// get unit number ----------------------------------------------------------
      L     DB1120.DBW    0;
      T     #UnitNo;

// communication ------------------------------------------------------------
      UC    FB  1125; // WT12Com

NETWORK
TITLE =Sequence organisation

      CLR   ;
      =     M    122.2;

// CIP Counter
      CALL FC    29 (
           UnitNo                   := #UnitNo,
           Value                    := DB1125.DBD   54,
           Enable                   := TRUE,
           Down                     := FALSE,
           OriginDetect             := 0.000000e+000,
           MaxDiffPS                := 1.000000e+000,
           SFMRec                   := DB1121.Seq.SFM[15],
           ValueOld                 := DB1121.DBD 1418);

// sequencer ----------------------------------------------------------------
      A     DB1123.DBX   43.1;
      S     DB1123.DBX   97.3;

      CALL FC    40 (
           UnitNo                   := #UnitNo);

END_FUNCTION_BLOCK

FUNCTION_BLOCK FB 1130
TITLE =U013: Wassertank 13
FAMILY : BOTEC_F1
NAME : U013A
VERSION : 2.1


VAR_TEMP
  EStopOK : BOOL ;	//auxiliary flag
  CIP : BOOL ;	//CIP Program Selected
  xTmp : BOOL ;	//Temporary Bool(free for general use)
  DummyBool : BOOL ;	//Temporary Bool(free for general use)
  UnitNo : INT ;	//unit number
  UnitFB : INT ;	//unit expansion FB number
  rTmp : REAL ;	//Temporary REAL (free for general use)
  iTmp : INT ;	//Temporary INT (free for general use)
  DummyInt : INT ;	//Temporary INT (free for general use)
  dTmp : DINT ;	//Temporary DINT (free for general use)
END_VAR
BEGIN
NETWORK
TITLE =general

      CLR   ;
      =     #xTmp;
      =     #EStopOK;

      L     DB1130.DBW    0;
      T     #UnitNo;
      L     DB1130.DBW    2;
      T     #UnitFB;

NETWORK
TITLE =analog inputs

      NOP   0;
// LI_T13 AnI 001 Niveau Tank 13
      CALL FC    24 (
           UnitNo                   := #UnitNo,
           AnIRec                   := DB2133.LI_T13,
           ValPer                   := DB302.DBW   88);

NETWORK
TITLE =Universal value

      NOP   0;
// unv001 UnV 001 Process Status
      CALL FC    27 (
           UnitNo                   := #UnitNo,
           UnVRec                   := DB2135.unv001,
           ValExt                   := DB2135.DBD  234);

// unv002 UnV 002 Universal Value 02
      CALL FC    27 (
           UnitNo                   := #UnitNo,
           UnVRec                   := DB2135.unv002,
           ValExt                   := DB2135.DBD  362);

// unv003 UnV 003 Universal Value 03
      CALL FC    27 (
           UnitNo                   := #UnitNo,
           UnVRec                   := DB2135.unv003,
           ValExt                   := DB2135.DBD  490);

NETWORK
TITLE =special inputs

      NOP   0;
// LS_LLL_T13 SpI 001 LS- Tank 13
      CALL FC    14 (
           UnitNo                   := #UnitNo,
           SpIRec                   := DB2131.LS_LLL_T13,
           SpIBit                   := I     50.0);

// LS_HL_T13 SpI 002 LS+ Tank 13
      CALL FC    14 (
           UnitNo                   := #UnitNo,
           SpIRec                   := DB2131.LS_HL_T13,
           SpIBit                   := I     49.6);

// GOA_T13_ML SpI 003 Mannloch Tank 13
      CALL FC    14 (
           UnitNo                   := #UnitNo,
           SpIRec                   := DB2131.GOA_T13_ML,
           SpIBit                   := I     49.5);

// GOA_T13_VV SpI 004 Vacuumventil Tank 13
      CALL FC    14 (
           UnitNo                   := #UnitNo,
           SpIRec                   := DB2131.GOA_T13_VV,
           SpIBit                   := I     49.4);

// LS_LL_T13 SpI 005 LS/ Tank 13
      CALL FC    14 (
           UnitNo                   := #UnitNo,
           SpIRec                   := DB2131.LS_LL_T13,
           SpIBit                   := I     49.7);

// RM_NI_T13_K4_AUF SpI 006
      CALL FC    14 (
           UnitNo                   := #UnitNo,
           SpIRec                   := DB2131.RM_NI_T13_K4_AUF,
           SpIBit                   := I     49.2);

// RM_NI_T13_K4_ZU SpI 007
      CALL FC    14 (
           UnitNo                   := #UnitNo,
           SpIRec                   := DB2131.RM_NI_T13_K4_ZU,
           SpIBit                   := I     49.3);

// RM_NI_T13_K2 SpI 008
      CALL FC    14 (
           UnitNo                   := #UnitNo,
           SpIRec                   := DB2131.RM_NI_T13_K2,
           SpIBit                   := I     49.0);

// RM_NI_T13_K3 SpI 010
      CALL FC    14 (
           UnitNo                   := #UnitNo,
           SpIRec                   := DB2131.RM_NI_T13_K3,
           SpIBit                   := I     49.1);

// LABOR_FREIG_T13 SpI 011 SCHLUESSELSCHALTER LABOR
      CALL FC    14 (
           UnitNo                   := #UnitNo,
           SpIRec                   := DB2131.LABOR_FREIG_T13,
           SpIBit                   := I    259.5);

NETWORK
TITLE =messages

      NOP   0;
// msg001 Msg 001 Message 01
      CALL FC    16 (
           UnitNo                   := #UnitNo,
           MsgRec                   := DB2137.msg001,
           MsgBit                   := DB2137.DBX   82.7);

// msg002 Msg 002 Message 02
      CALL FC    16 (
           UnitNo                   := #UnitNo,
           MsgRec                   := DB2137.msg002,
           MsgBit                   := DB2137.DBX  142.7);

NETWORK
TITLE =unit supply

      UC    FB [#UnitFB];

NETWORK
TITLE =T13_A10
// Act 005
// Box           : Ventilinsel 2
// Input address : I317.4
// Output address: Q317.4
      CALL FC    70 (
           UnitNo                   := #UnitNo,
           ActRec                   := DB2130.T13_A10,
           Typ                      := 1,
           FBa                      := #xTmp,
           FBa2                     := I    317.4,
           Out                      := Q    317.4);

NETWORK
TITLE =T13_A9
// Act 006
// Box           : Ventilinsel 2
// Input address : I319.4
// Output address: Q319.4
      CALL FC    70 (
           UnitNo                   := #UnitNo,
           ActRec                   := DB2130.T13_A9,
           Typ                      := 1,
           FBa                      := #xTmp,
           FBa2                     := I    319.4,
           Out                      := Q    319.4);

NETWORK
TITLE =T13_A12
// Act 007
// Box           : Ventilinsel 2
// Input address : I321.4
// Output address: Q321.4
      CALL FC    70 (
           UnitNo                   := #UnitNo,
           ActRec                   := DB2130.T13_A12,
           Typ                      := 1,
           FBa                      := #xTmp,
           FBa2                     := I    321.4,
           Out                      := Q    321.4);

NETWORK
TITLE =T13_A7
// Act 008
// Box           : Ventilinsel 2
// Input address : I323.4
// Output address: Q323.4
      CALL FC    70 (
           UnitNo                   := #UnitNo,
           ActRec                   := DB2130.T13_A7,
           Typ                      := 1,
           FBa                      := #xTmp,
           FBa2                     := I    323.4,
           Out                      := Q    323.4);

NETWORK
TITLE =T13_A8
// Act 009
// Box           : Ventilinsel 3
// Input address : I325.4
// Output address: Q325.4
      CALL FC    70 (
           UnitNo                   := #UnitNo,
           ActRec                   := DB2130.T13_A8,
           Typ                      := 1,
           FBa                      := #xTmp,
           FBa2                     := I    325.4,
           Out                      := Q    325.4);

NETWORK
TITLE =T13_A5
// Act 010
// Box           : Ventilinsel 3
// Input address : I327.4
// Output address: Q327.4
      CALL FC    70 (
           UnitNo                   := #UnitNo,
           ActRec                   := DB2130.T13_A5,
           Typ                      := 1,
           FBa                      := #xTmp,
           FBa2                     := I    327.4,
           Out                      := Q    327.4);

NETWORK
TITLE =T13_A11
// Act 011
// Box           : Ventilinsel 3
// Input address : I329.4
// Output address: Q329.4
      CALL FC    70 (
           UnitNo                   := #UnitNo,
           ActRec                   := DB2130.T13_A11,
           Typ                      := 1,
           FBa                      := #xTmp,
           FBa2                     := I    329.4,
           Out                      := Q    329.4);

NETWORK
TITLE =T13_A14
// Act 012
// Box           : Ventilinsel 4
// Input address : I331.4
// Output address: Q331.4
      CALL FC    70 (
           UnitNo                   := #UnitNo,
           ActRec                   := DB2130.T13_A14,
           Typ                      := 1,
           FBa                      := #xTmp,
           FBa2                     := I    331.4,
           Out                      := Q    331.4);

NETWORK
TITLE =T13_A15
// Act 013
// Box           : Ventilinsel 4
// Input address : I333.4
// Output address: Q333.4
      CALL FC    70 (
           UnitNo                   := #UnitNo,
           ActRec                   := DB2130.T13_A15,
           Typ                      := 0,
           FBa                      := #xTmp,
           FBa2                     := I    333.4,
           Out                      := Q    333.4);

NETWORK
TITLE =T13_RR1
// Act 014
// Box           : Ventilinsel 4
// Input address : I335.4
// Output address: Q335.4
      CALL FC    70 (
           UnitNo                   := #UnitNo,
           ActRec                   := DB2130.T13_RR1,
           Typ                      := 1,
           FBa                      := #xTmp,
           FBa2                     := I    335.4,
           Out                      := Q    335.4);

NETWORK
TITLE =RV1_T13
// Act 015
// Box           : Ventilinsel 1
// Input address : I10.4
// Output address: Q10.4
      CALL FC    70 (
           UnitNo                   := #UnitNo,
           ActRec                   := DB2130.RV1_T13,
           Typ                      := 1,
           FBa                      := #xTmp,
           FBa2                     := I     10.4,
           Out                      := Q     10.4);

NETWORK
TITLE =B6F_T13
// Act 016
// Box           : Ventilinsel 1
// Input address : I10.5
// Output address: Q10.5
      CALL FC    70 (
           UnitNo                   := #UnitNo,
           ActRec                   := DB2130.B6F_T13,
           Typ                      := 1,
           FBa                      := #xTmp,
           FBa2                     := I     10.5,
           Out                      := Q     10.5);

NETWORK
TITLE =H6F_T13
// Act 017
// Box           : Ventilinsel 1
// Input address : I10.6
// Output address: Q10.6
      CALL FC    70 (
           UnitNo                   := #UnitNo,
           ActRec                   := DB2130.H6F_T13,
           Typ                      := 1,
           FBa                      := #xTmp,
           FBa2                     := I     10.6,
           Out                      := Q     10.6);

NETWORK
TITLE =J6F_T13
// Act 018
// Box           : Ventilinsel 1
// Input address : I10.7
// Output address: Q10.7
      CALL FC    70 (
           UnitNo                   := #UnitNo,
           ActRec                   := DB2130.J6F_T13,
           Typ                      := 1,
           FBa                      := #xTmp,
           FBa2                     := I     10.7,
           Out                      := Q     10.7);

NETWORK
TITLE =L6F_T13
// Act 019
// Box           : Ventilinsel 1
// Input address : I11.0
// Output address: Q11.0
      CALL FC    70 (
           UnitNo                   := #UnitNo,
           ActRec                   := DB2130.L6F_T13,
           Typ                      := 1,
           FBa                      := #xTmp,
           FBa2                     := I     11.0,
           Out                      := Q     11.0);

NETWORK
TITLE =A_T13
// Act 022
// Box           : Ventilinsel 1
// Input address : I11.3
// Output address: Q11.3
      CALL FC    70 (
           UnitNo                   := #UnitNo,
           ActRec                   := DB2130.A_T13,
           Typ                      := 1,
           FBa                      := #xTmp,
           FBa2                     := I     11.3,
           Out                      := Q     11.3);

NETWORK
TITLE =B_T13
// Act 023
// Box           : Ventilinsel 1
// Input address : I11.4
// Output address: Q11.4
      CALL FC    70 (
           UnitNo                   := #UnitNo,
           ActRec                   := DB2130.B_T13,
           Typ                      := 1,
           FBa                      := #xTmp,
           FBa2                     := I     11.4,
           Out                      := Q     11.4);

NETWORK
TITLE =RW5_T13
// Act 026
// Box           : Ventilinsel 1
// Input address : I11.6
// Output address: Q11.6
      CALL FC    70 (
           UnitNo                   := #UnitNo,
           ActRec                   := DB2130.RW5_T13,
           Typ                      := 1,
           FBa                      := #xTmp,
           FBa2                     := I     11.6,
           Out                      := Q     11.6);

NETWORK
TITLE =RW6_T13
// Act 027
// Box           : Ventilinsel 1
// Input address : I11.7
// Output address: Q11.7
      CALL FC    70 (
           UnitNo                   := #UnitNo,
           ActRec                   := DB2130.RW6_T13,
           Typ                      := 1,
           FBa                      := #xTmp,
           FBa2                     := I     11.7,
           Out                      := Q     11.7);

NETWORK
TITLE =VVT13  Vacuumventil Tank 13
// Act 028
// Box           : VST1-9
// Output address: Q160.2
      CALL FC    70 (
           UnitNo                   := #UnitNo,
           ActRec                   := DB2130.VVT13,
           Typ                      := 0,
           FBa                      := #xTmp,
           FBa2                     := #xTmp,
           Out                      := Q    160.2);

NETWORK
TITLE =VR_T13
// Act 029
// Box           : Ventilinsel 1
// Output address: Q11.5
      CALL FC    70 (
           UnitNo                   := #UnitNo,
           ActRec                   := DB2130.VR_T13,
           Typ                      := 0,
           FBa                      := #xTmp,
           FBa2                     := #xTmp,
           Out                      := Q     11.5);

NETWORK
TITLE =ML_LABORFREIGABE_T13
// Act 031
// Box           : LT-CIP
// Output address: Q259.5
      CALL FC    70 (
           UnitNo                   := #UnitNo,
           ActRec                   := DB2130.ML_LABORFREIGABE_T13,
           Typ                      := 0,
           FBa                      := #xTmp,
           FBa2                     := #xTmp,
           Out                      := Q    259.5);

END_FUNCTION_BLOCK

FUNCTION_BLOCK FB 1131
TITLE =U013: Water Tank 13
FAMILY : BOTEC_F1
NAME : UniE
VERSION : 1.2


VAR_TEMP
  CIP : BOOL ;	//CIP active
  UNIM : BOOL ;	//Unit Not In Maintenance
  GenRel : BOOL ;	//general OK (emergency and maintenance OK)
  EStopOK : BOOL ;	//emergency OK
  UnitNo : INT ;	//unit number
  xTmp : BOOL ;	//Temporary Bool
  iTmp : INT ;	//Temporary INT
  rTmp : REAL ;	//Temporary REAL
  dTmp : DINT ;	//Temporary DINT (free for general use)
  RetValInt : INT ;	//return value
END_VAR
BEGIN
NETWORK
TITLE =General

      SET   ;
// Simulation ---------------------------------------------------------------
      A     DB1131.DBX 1357.7;
      CC    FB  1139; // "WT13Sim"
      A     DB1131.DBX   17.3;
      =     DB1131.DBX 1357.7; //Help bit for simulation

// get unit number ----------------------------------------------------------
      L     DB1130.DBW    0;
      T     #UnitNo;

// communication ------------------------------------------------------------
      UC    FB  1135; // WT13Com

NETWORK
TITLE =Sequence organisation

      CLR   ;
      =     M    122.2;

// CIP Counter
      CALL FC    29 (
           UnitNo                   := #UnitNo,
           Value                    := DB1135.DBD   54,
           Enable                   := TRUE,
           Down                     := FALSE,
           OriginDetect             := 0.000000e+000,
           MaxDiffPS                := 1.000000e+000,
           SFMRec                   := DB1131.Seq.SFM[15],
           ValueOld                 := DB1131.DBD 1418);

// sequencer ----------------------------------------------------------------
      A     DB1133.DBX   43.1;
      S     DB1133.DBX   97.3;

      CALL FC    40 (
           UnitNo                   := #UnitNo);

END_FUNCTION_BLOCK

FUNCTION_BLOCK FB 1210
TITLE =U021: Brunnen Transfer VE1
FAMILY : BOTEC_F1
NAME : U021A
VERSION : 2.1


VAR_TEMP
  EStopOK : BOOL ;	//auxiliary flag
  CIP : BOOL ;	//CIP Program Selected
  xTmp : BOOL ;	//Temporary Bool(free for general use)
  DummyBool : BOOL ;	//Temporary Bool(free for general use)
  UnitNo : INT ;	//unit number
  UnitFB : INT ;	//unit expansion FB number
  rTmp : REAL ;	//Temporary REAL (free for general use)
  iTmp : INT ;	//Temporary INT (free for general use)
  DummyInt : INT ;	//Temporary INT (free for general use)
  dTmp : DINT ;	//Temporary DINT (free for general use)
END_VAR
BEGIN
NETWORK
TITLE =general

      CLR   ;
      =     #xTmp;
      =     #EStopOK;

      L     DB1210.DBW    0;
      T     #UnitNo;
      L     DB1210.DBW    2;
      T     #UnitFB;

NETWORK
TITLE =analog inputs

      NOP   0;
// C_AnI01 AnI 001 spare
      CALL FC    24 (
           UnitNo                   := #UnitNo,
           AnIRec                   := DB2213.C_AnI01,
           ValPer                   := #DummyInt);

// C_AnI002 AnI 002 spare
      CALL FC    24 (
           UnitNo                   := #UnitNo,
           AnIRec                   := DB2213.C_AnI002,
           ValPer                   := #DummyInt);

// AnI03 AnI 003 spare
      CALL FC    24 (
           UnitNo                   := #UnitNo,
           AnIRec                   := DB2213.AnI03,
           ValPer                   := #DummyInt);

NETWORK
TITLE =Universal value

      NOP   0;
// unv001 UnV 001 Process Status
      CALL FC    27 (
           UnitNo                   := #UnitNo,
           UnVRec                   := DB2215.unv001,
           ValExt                   := DB2215.DBD  234);

// unv002 UnV 002 Universal Value 02
      CALL FC    27 (
           UnitNo                   := #UnitNo,
           UnVRec                   := DB2215.unv002,
           ValExt                   := DB2215.DBD  362);

// unv003 UnV 003 Universal Value 03
      CALL FC    27 (
           UnitNo                   := #UnitNo,
           UnVRec                   := DB2215.unv003,
           ValExt                   := DB2215.DBD  490);

// unv004 UnV 004 Universal Value 04
      CALL FC    27 (
           UnitNo                   := #UnitNo,
           UnVRec                   := DB2215.unv004,
           ValExt                   := DB2215.DBD  618);

NETWORK
TITLE =special inputs

      NOP   0;
// NI_VP1_Br2a_VE1 SpI 001 Paneel VP1 Brunnen 2a -> VE1
      CALL FC    14 (
           UnitNo                   := #UnitNo,
           SpIRec                   := DB2211.NI_VP1_Br2a_VE1,
           SpIBit                   := I     80.1);

// NI_VP1_Br2b_VE1 SpI 002 Paneel VP1 Brunnen 2b -> VE1
      CALL FC    14 (
           UnitNo                   := #UnitNo,
           SpIRec                   := DB2211.NI_VP1_Br2b_VE1,
           SpIBit                   := I     80.2);

// NI_VP1_Br3_VE1 SpI 003 Paneel VP1 Brunnen 3 -> VE1
      CALL FC    14 (
           UnitNo                   := #UnitNo,
           SpIRec                   := DB2211.NI_VP1_Br3_VE1,
           SpIBit                   := I     80.4);

// NI_VP1_Br7_VE1 SpI 004 Paneel VP1 Brunnen 7 -> VE1
      CALL FC    14 (
           UnitNo                   := #UnitNo,
           SpIRec                   := DB2211.NI_VP1_Br7_VE1,
           SpIBit                   := I     80.3);

NETWORK
TITLE =messages

      NOP   0;
// msg001 Msg 001 Message 01
      CALL FC    16 (
           UnitNo                   := #UnitNo,
           MsgRec                   := DB2217.msg001,
           MsgBit                   := DB2217.DBX   82.7);

// msg002 Msg 002 Message 02
      CALL FC    16 (
           UnitNo                   := #UnitNo,
           MsgRec                   := DB2217.msg002,
           MsgBit                   := DB2217.DBX  142.7);

// msg003 Msg 003 Message 03
      CALL FC    16 (
           UnitNo                   := #UnitNo,
           MsgRec                   := DB2217.msg003,
           MsgBit                   := DB2217.DBX  202.7);

NETWORK
TITLE =controllers

      NOP   0;
// PID01 PID 001 spare
      CALL FC    55 (
           UnitNo                   := #UnitNo,
           PIDRec                   := DB2216.PID01,
           SpExt                    := DB2216.DBD  234,
           PVal                     := DB2216.DBD  254,
           OPer                     := #DummyInt);

NETWORK
TITLE =unit supply

      UC    FB [#UnitFB];

NETWORK
TITLE =RW6_G1  Gullyventil RW6
// Act 001
// Box           : VS2-BB
// Input address : I310.4
// Output address: Q310.4
      CALL FC    70 (
           UnitNo                   := #UnitNo,
           ActRec                   := DB2210.RW6_G1,
           Typ                      := 1,
           FBa                      := #xTmp,
           FBa2                     := I    310.4,
           Out                      := Q    310.4);

NETWORK
TITLE =VE1V1  VE1V1 --> Chriwa
// Act 002
// Box           : VS2-BB
// Input address : I310.5
// Output address: Q310.5
      CALL FC    70 (
           UnitNo                   := #UnitNo,
           ActRec                   := DB2210.VE1V1,
           Typ                      := 23,
           FBa                      := I    310.5,
           FBa2                     := #xTmp,
           Out                      := Q    310.5);

NETWORK
TITLE =VE1V2  VE1V2 Gully
// Act 003
// Box           : VS2-BB
// Input address : I310.6
// Output address: Q310.6
      CALL FC    70 (
           UnitNo                   := #UnitNo,
           ActRec                   := DB2210.VE1V2,
           Typ                      := 1,
           FBa                      := #xTmp,
           FBa2                     := I    310.6,
           Out                      := Q    310.6);

END_FUNCTION_BLOCK

FUNCTION_BLOCK FB 1211
TITLE =U021: Well Transfer VE1
FAMILY : BOTEC_F1
NAME : UniE
VERSION : 1.2


VAR_TEMP
  CIP : BOOL ;	//CIP active
  UNIM : BOOL ;	//Unit Not In Maintenance
  GenRel : BOOL ;	//general OK (emergency and maintenance OK)
  EStopOK : BOOL ;	//emergency OK
  UnitNo : INT ;	//unit number
  xTmp : BOOL ;	//Temporary Bool
  iTmp : INT ;	//Temporary INT
  rTmp : REAL ;	//Temporary REAL
  dTmp : DINT ;	//Temporary DINT (free for general use)
  RetValInt : INT ;	//return value
END_VAR
BEGIN
NETWORK
TITLE =General

      SET   ;
// Simulation ---------------------------------------------------------------
      A     DB1211.DBX 1357.7;
      CC    FB  1219; // "U021Sim"
      A     DB1211.DBX   17.3;
      =     DB1211.DBX 1357.7; //Help bit for simulation

// get unit number ----------------------------------------------------------
      L     DB1210.DBW    0;
      T     #UnitNo;

// communication ------------------------------------------------------------
      UC    FB  1215; // U021Com

NETWORK
TITLE =Sequence organisation

      CLR   ;
      =     M    122.2;


// Chriwa Status 1
      L     DB1381.DBD  482;
      T     DB1211.DBD  482;

// Chriwa Status 2
      L     DB1381.DBD  498;
      T     DB1211.DBD  498;

// sequencer ----------------------------------------------------------------
      A     DB1213.DBX   43.1;
      S     DB1213.DBX   97.3;

      CALL FC    40 (
           UnitNo                   := #UnitNo);

END_FUNCTION_BLOCK

FUNCTION_BLOCK FB 1220
TITLE =U022: Brunnen Transfer VE2
FAMILY : BOTEC_F1
NAME : U022A
VERSION : 2.1


VAR_TEMP
  EStopOK : BOOL ;	//auxiliary flag
  CIP : BOOL ;	//CIP Program Selected
  xTmp : BOOL ;	//Temporary Bool(free for general use)
  DummyBool : BOOL ;	//Temporary Bool(free for general use)
  UnitNo : INT ;	//unit number
  UnitFB : INT ;	//unit expansion FB number
  rTmp : REAL ;	//Temporary REAL (free for general use)
  iTmp : INT ;	//Temporary INT (free for general use)
  DummyInt : INT ;	//Temporary INT (free for general use)
  dTmp : DINT ;	//Temporary DINT (free for general use)
END_VAR
BEGIN
NETWORK
TITLE =general

      CLR   ;
      =     #xTmp;
      =     #EStopOK;

      L     DB1220.DBW    0;
      T     #UnitNo;
      L     DB1220.DBW    2;
      T     #UnitFB;

NETWORK
TITLE =analog inputs

      NOP   0;
// C_AnI01 AnI 001 spare
      CALL FC    24 (
           UnitNo                   := #UnitNo,
           AnIRec                   := DB2223.C_AnI01,
           ValPer                   := #DummyInt);

// C_AnI002 AnI 002 spare
      CALL FC    24 (
           UnitNo                   := #UnitNo,
           AnIRec                   := DB2223.C_AnI002,
           ValPer                   := #DummyInt);

// AnI03 AnI 003 spare
      CALL FC    24 (
           UnitNo                   := #UnitNo,
           AnIRec                   := DB2223.AnI03,
           ValPer                   := #DummyInt);

NETWORK
TITLE =Universal value

      NOP   0;
// unv001 UnV 001 Process Status
      CALL FC    27 (
           UnitNo                   := #UnitNo,
           UnVRec                   := DB2225.unv001,
           ValExt                   := DB2225.DBD  234);

// unv002 UnV 002 Universal Value 02
      CALL FC    27 (
           UnitNo                   := #UnitNo,
           UnVRec                   := DB2225.unv002,
           ValExt                   := DB2225.DBD  362);

// unv003 UnV 003 Universal Value 03
      CALL FC    27 (
           UnitNo                   := #UnitNo,
           UnVRec                   := DB2225.unv003,
           ValExt                   := DB2225.DBD  490);

// unv004 UnV 004 Universal Value 04
      CALL FC    27 (
           UnitNo                   := #UnitNo,
           UnVRec                   := DB2225.unv004,
           ValExt                   := DB2225.DBD  618);

NETWORK
TITLE =special inputs

      NOP   0;
// NI_VP1_Br2a_VE2 SpI 001 Paneel VP1 Brunnen 2a -> VE2
      CALL FC    14 (
           UnitNo                   := #UnitNo,
           SpIRec                   := DB2221.NI_VP1_Br2a_VE2,
           SpIBit                   := I     80.6);

// NI_VP1_Br2b_VE2 SpI 002 Paneel VP1 Brunnen 2b -> VE2
      CALL FC    14 (
           UnitNo                   := #UnitNo,
           SpIRec                   := DB2221.NI_VP1_Br2b_VE2,
           SpIBit                   := I     80.7);

// NI_VP1_Br3_VE2 SpI 003 Paneel VP1 Brunnen 3 -> VE2
      CALL FC    14 (
           UnitNo                   := #UnitNo,
           SpIRec                   := DB2221.NI_VP1_Br3_VE2,
           SpIBit                   := I     81.1);

// NI_VP1_Br7_VE2 SpI 004 Paneel VP1 Brunnen 7 -> VE2
      CALL FC    14 (
           UnitNo                   := #UnitNo,
           SpIRec                   := DB2221.NI_VP1_Br7_VE2,
           SpIBit                   := I     81.0);

NETWORK
TITLE =messages

      NOP   0;
// msg001 Msg 001 Message 01
      CALL FC    16 (
           UnitNo                   := #UnitNo,
           MsgRec                   := DB2227.msg001,
           MsgBit                   := DB2227.DBX   82.7);

// msg002 Msg 002 Message 02
      CALL FC    16 (
           UnitNo                   := #UnitNo,
           MsgRec                   := DB2227.msg002,
           MsgBit                   := DB2227.DBX  142.7);

// msg003 Msg 003 Message 03
      CALL FC    16 (
           UnitNo                   := #UnitNo,
           MsgRec                   := DB2227.msg003,
           MsgBit                   := DB2227.DBX  202.7);

NETWORK
TITLE =controllers

      NOP   0;
// PID01 PID 001 spare
      CALL FC    55 (
           UnitNo                   := #UnitNo,
           PIDRec                   := DB2226.PID01,
           SpExt                    := DB2226.DBD  234,
           PVal                     := DB2226.DBD  254,
           OPer                     := #DummyInt);

NETWORK
TITLE =unit supply

      UC    FB [#UnitFB];

NETWORK
TITLE =RW5_G1  Gullyventil RW5
// Act 001
// Box           : VS2-BB
// Input address : I310.3
// Output address: Q310.3
      CALL FC    70 (
           UnitNo                   := #UnitNo,
           ActRec                   := DB2220.RW5_G1,
           Typ                      := 1,
           FBa                      := #xTmp,
           FBa2                     := I    310.3,
           Out                      := Q    310.3);

NETWORK
TITLE =VE2V1  VE2V1 --> Chriwa
// Act 002
// Box           : VS2-BB
// Input address : I310.7
// Output address: Q310.7
      CALL FC    70 (
           UnitNo                   := #UnitNo,
           ActRec                   := DB2220.VE2V1,
           Typ                      := 23,
           FBa                      := I    310.7,
           FBa2                     := #xTmp,
           Out                      := Q    310.7);

NETWORK
TITLE =VE2V2  VE2V2 Gully
// Act 003
// Box           : VS2-BB
// Input address : I311.0
// Output address: Q311.0
      CALL FC    70 (
           UnitNo                   := #UnitNo,
           ActRec                   := DB2220.VE2V2,
           Typ                      := 1,
           FBa                      := #xTmp,
           FBa2                     := I    311.0,
           Out                      := Q    311.0);

END_FUNCTION_BLOCK

FUNCTION_BLOCK FB 1221
TITLE =U022: Well Transfer VE2
FAMILY : BOTEC_F1
NAME : UniE
VERSION : 1.2


VAR_TEMP
  CIP : BOOL ;	//CIP active
  UNIM : BOOL ;	//Unit Not In Maintenance
  GenRel : BOOL ;	//general OK (emergency and maintenance OK)
  EStopOK : BOOL ;	//emergency OK
  UnitNo : INT ;	//unit number
  xTmp : BOOL ;	//Temporary Bool
  iTmp : INT ;	//Temporary INT
  rTmp : REAL ;	//Temporary REAL
  dTmp : DINT ;	//Temporary DINT (free for general use)
  RetValInt : INT ;	//return value
END_VAR
BEGIN
NETWORK
TITLE =General

      SET   ;
// Simulation ---------------------------------------------------------------
      A     DB1221.DBX 1357.7;
      CC    FB  1229; // "U022Sim"
      A     DB1221.DBX   17.3;
      =     DB1221.DBX 1357.7; //Help bit for simulation

// get unit number ----------------------------------------------------------
      L     DB1220.DBW    0;
      T     #UnitNo;

// communication ------------------------------------------------------------
      UC    FB  1225; // U022Com

NETWORK
TITLE =Sequence organisation

      CLR   ;
      =     M    122.2;


// Chriwa Status 1
      L     DB1391.DBD  482;
      T     DB1221.DBD  482;

// Chriwa Status 2
      L     DB1391.DBD  498;
      T     DB1221.DBD  498;

// sequencer ----------------------------------------------------------------
      A     DB1223.DBX   43.1;
      S     DB1223.DBX   97.3;

      CALL FC    40 (
           UnitNo                   := #UnitNo);

END_FUNCTION_BLOCK

FUNCTION_BLOCK FB 1250
TITLE =U025: Well Transfer A
FAMILY : BOTEC_F1
NAME : UniA
VERSION : 2.1


VAR_TEMP
  EStopOK : BOOL ;	//auxiliary flag
  CIP : BOOL ;	//CIP Program Selected
  xTmp : BOOL ;	//Temporary Bool(free for general use)
  UnitNo : INT ;	//unit number
  UnitFB : INT ;	//unit expansion FB number
  rTmp : REAL ;	//Temporary REAL (free for general use)
  iTmp : INT ;	//Temporary INT (free for general use)
  dTmp : DINT ;	//Temporary DINT (free for general use)
END_VAR
BEGIN
NETWORK
TITLE =general

      CLR   ;
      =     #xTmp;
      =     #EStopOK;

      L     DB1250.DBW    0;
      T     #UnitNo;
      L     DB1250.DBW    2;
      T     #UnitFB;

NETWORK
TITLE =analog inputs

      NOP   0;
// C_AnI01 AnI 001 spare
      CALL FC    24 (
           UnitNo                   := #UnitNo,
           AnIRec                   := DB2253.C_AnI01,
           ValPer                   := #iTmp);

// QI_CO2_A_PH AnI 002
      CALL FC    24 (
           UnitNo                   := #UnitNo,
           AnIRec                   := DB2253.QI_CO2_A_PH,
           ValPer                   := IW   220);

// QI_CO2_A_pH_KOR AnI 003 pH Brunnen A mit Offset
      CALL FC    24 (
           UnitNo                   := #UnitNo,
           AnIRec                   := DB2253.QI_CO2_A_pH_KOR,
           ValPer                   := IW   552);

NETWORK
TITLE =Universal value

      NOP   0;
// unv001 UnV 001 Process Status
      CALL FC    27 (
           UnitNo                   := #UnitNo,
           UnVRec                   := DB2255.unv001,
           ValExt                   := DB2255.DBD  234);

// unv002 UnV 002 Universal Value 02
      CALL FC    27 (
           UnitNo                   := #UnitNo,
           UnVRec                   := DB2255.unv002,
           ValExt                   := DB2255.DBD  362);

// unv003 UnV 003 Universal Value 03
      CALL FC    27 (
           UnitNo                   := #UnitNo,
           UnVRec                   := DB2255.unv003,
           ValExt                   := DB2255.DBD  490);

// unv004 UnV 004 Universal Value 04
      CALL FC    27 (
           UnitNo                   := #UnitNo,
           UnVRec                   := DB2255.unv004,
           ValExt                   := DB2255.DBD  618);

NETWORK
TITLE =special inputs

      NOP   0;
// SpI01 SpI 001 spare
      CALL FC    14 (
           UnitNo                   := #UnitNo,
           SpIRec                   := DB2251.SpI01,
           SpIBit                   := #xTmp);

// SpI02 SpI 002 spare
      CALL FC    14 (
           UnitNo                   := #UnitNo,
           SpIRec                   := DB2251.SpI02,
           SpIBit                   := #xTmp);

// SpI03 SpI 003 spare
      CALL FC    14 (
           UnitNo                   := #UnitNo,
           SpIRec                   := DB2251.SpI03,
           SpIBit                   := #xTmp);

// SpI04 SpI 004 spare
      CALL FC    14 (
           UnitNo                   := #UnitNo,
           SpIRec                   := DB2251.SpI04,
           SpIBit                   := #xTmp);

NETWORK
TITLE =messages

      NOP   0;
// msg001 Msg 001 Message 01
      CALL FC    16 (
           UnitNo                   := #UnitNo,
           MsgRec                   := DB2257.msg001,
           MsgBit                   := DB2257.DBX   82.7);

// msg002 Msg 002 Message 02
      CALL FC    16 (
           UnitNo                   := #UnitNo,
           MsgRec                   := DB2257.msg002,
           MsgBit                   := DB2257.DBX  142.7);

// msg003 Msg 003 Message 03
      CALL FC    16 (
           UnitNo                   := #UnitNo,
           MsgRec                   := DB2257.msg003,
           MsgBit                   := DB2257.DBX  202.7);

NETWORK
TITLE =controllers

      NOP   0;
// CO2ARV1 PID 001 CO2 A RV1
      CALL FC    55 (
           UnitNo                   := #UnitNo,
           PIDRec                   := DB2256.CO2ARV1,
           SpExt                    := DB2256.DBD  234,
           PVal                     := DB2256.DBD  254,
           OPer                     := PQW  220);

NETWORK
TITLE =unit supply

      UC    FB [#UnitFB];

NETWORK
TITLE =A_G1  A_G1
// Act 001
// Box           : VS2-BB
// Output address: Q309.3
      CALL FC    70 (
           UnitNo                   := #UnitNo,
           ActRec                   := DB2250.A_G1,
           Typ                      := 1,
           FBa                      := #xTmp,
           FBa2                     := I    309.3,
           Out                      := Q    309.3);

NETWORK
TITLE =CO2_AV2  Ansteuerung AV2
// Act 002
// Box           : CO2 Dosierung
// Output address: Q61.7
      CALL FC    70 (
           UnitNo                   := #UnitNo,
           ActRec                   := DB2250.CO2_AV2,
           Typ                      := 0,
           FBa                      := #xTmp,
           FBa2                     := #xTmp,
           Out                      := Q     61.7);

NETWORK
TITLE =CO2_AV1  Ansteuerung AV1
// Act 003
// Box           : CO2 Dosierung
// Output address: Q60.7
      CALL FC    70 (
           UnitNo                   := #UnitNo,
           ActRec                   := DB2250.CO2_AV1,
           Typ                      := 0,
           FBa                      := #xTmp,
           FBa2                     := #xTmp,
           Out                      := Q     60.7);

NETWORK
TITLE =ARV1  CO2 A RV1
// Act 004
// Box           :
// Input address : #xtmp
// Output address: #xtmp
      CALL FC    70 (
           UnitNo                   := #UnitNo,
           ActRec                   := DB2250.ARV1,
           Typ                      := 4,
           FBa                      := #xTmp,
           FBa2                     := #xTmp,
           Out                      := #xTmp);

END_FUNCTION_BLOCK

FUNCTION_BLOCK FB 1251
TITLE =U025: Well Transfer A
FAMILY : BOTEC_F1
NAME : UniE
VERSION : 1.2


VAR_TEMP
  CIP : BOOL ;	//CIP active
  UNIM : BOOL ;	//Unit Not In Maintenance
  GenRel : BOOL ;	//general OK (emergency and maintenance OK)
  EStopOK : BOOL ;	//emergency OK
  UnitNo : INT ;	//unit number
  xTmp : BOOL ;	//Temporary Bool
  iTmp : INT ;	//Temporary INT
  rTmp : REAL ;	//Temporary REAL
  dTmp : DINT ;	//Temporary DINT (free for general use)
  RetValInt : INT ;	//return value
END_VAR
BEGIN
NETWORK
TITLE =General

      SET   ;
// Simulation ---------------------------------------------------------------
      A     DB1251.DBX 1357.7;
      CC    FB  1259; // "U025Sim"
      A     DB1251.DBX   17.3;
      =     DB1251.DBX 1357.7; //Help bit for simulation

// get unit number ----------------------------------------------------------
      L     DB1250.DBW    0;
      T     #UnitNo;

// communication ------------------------------------------------------------
      UC    FB  1255; // U025Com

NETWORK
TITLE =Sequence organisation

      CLR   ;
      =     M    122.2;

// sequencer ----------------------------------------------------------------
      A     DB1253.DBX   43.1;
      S     DB1253.DBX   97.3;

      CALL FC    40 (
           UnitNo                   := #UnitNo);

END_FUNCTION_BLOCK

FUNCTION_BLOCK FB 1260
TITLE =U026: Well Transfer B
FAMILY : BOTEC_F1
NAME : UniA
VERSION : 2.1


VAR_TEMP
  EStopOK : BOOL ;	//auxiliary flag
  CIP : BOOL ;	//CIP Program Selected
  xTmp : BOOL ;	//Temporary Bool(free for general use)
  UnitNo : INT ;	//unit number
  UnitFB : INT ;	//unit expansion FB number
  rTmp : REAL ;	//Temporary REAL (free for general use)
  iTmp : INT ;	//Temporary INT (free for general use)
  dTmp : DINT ;	//Temporary DINT (free for general use)
END_VAR
BEGIN
NETWORK
TITLE =general

      CLR   ;
      =     #xTmp;
      =     #EStopOK;

      L     DB1260.DBW    0;
      T     #UnitNo;
      L     DB1260.DBW    2;
      T     #UnitFB;

NETWORK
TITLE =analog inputs

      NOP   0;
// C_AnI01 AnI 001 spare
      CALL FC    24 (
           UnitNo                   := #UnitNo,
           AnIRec                   := DB2263.C_AnI01,
           ValPer                   := #iTmp);

// QI_CO2_B_PH AnI 002
      CALL FC    24 (
           UnitNo                   := #UnitNo,
           AnIRec                   := DB2263.QI_CO2_B_PH,
           ValPer                   := IW   222);

// AnI03 AnI 003 spare
      CALL FC    24 (
           UnitNo                   := #UnitNo,
           AnIRec                   := DB2263.AnI03,
           ValPer                   := #iTmp);

NETWORK
TITLE =Universal value

      NOP   0;
// unv001 UnV 001 Process Status
      CALL FC    27 (
           UnitNo                   := #UnitNo,
           UnVRec                   := DB2265.unv001,
           ValExt                   := DB2265.DBD  234);

// unv002 UnV 002 Universal Value 02
      CALL FC    27 (
           UnitNo                   := #UnitNo,
           UnVRec                   := DB2265.unv002,
           ValExt                   := DB2265.DBD  362);

// unv003 UnV 003 Universal Value 03
      CALL FC    27 (
           UnitNo                   := #UnitNo,
           UnVRec                   := DB2265.unv003,
           ValExt                   := DB2265.DBD  490);

// unv004 UnV 004 Universal Value 04
      CALL FC    27 (
           UnitNo                   := #UnitNo,
           UnVRec                   := DB2265.unv004,
           ValExt                   := DB2265.DBD  618);

NETWORK
TITLE =special inputs

      NOP   0;
// RM_NI_KF1_K1 SpI 001
      CALL FC    14 (
           UnitNo                   := #UnitNo,
           SpIRec                   := DB2261.RM_NI_KF1_K1,
           SpIBit                   := #xTmp);//"RM_NI_KF1_K1"

// RM_NI_KF1_K2 SpI 002
      CALL FC    14 (
           UnitNo                   := #UnitNo,
           SpIRec                   := DB2261.RM_NI_KF1_K2,
           SpIBit                   := #xTmp);//"RM_NI_KF1_K2"

// RM_NI_KF1_K3 SpI 003 PANEEL PTV1
      CALL FC    14 (
           UnitNo                   := #UnitNo,
           SpIRec                   := DB2261.RM_NI_KF1_K3,
           SpIBit                   := I     54.6);


// SpI04 SpI 004 spare
      CALL FC    14 (
           UnitNo                   := #UnitNo,
           SpIRec                   := DB2261.SpI04,
           SpIBit                   := #xTmp);

NETWORK
TITLE =messages

      NOP   0;
// msg001 Msg 001 Message 01
      CALL FC    16 (
           UnitNo                   := #UnitNo,
           MsgRec                   := DB2267.msg001,
           MsgBit                   := DB2267.DBX   82.7);

// msg002 Msg 002 Message 02
      CALL FC    16 (
           UnitNo                   := #UnitNo,
           MsgRec                   := DB2267.msg002,
           MsgBit                   := DB2267.DBX  142.7);

// msg003 Msg 003 Message 03
      CALL FC    16 (
           UnitNo                   := #UnitNo,
           MsgRec                   := DB2267.msg003,
           MsgBit                   := DB2267.DBX  202.7);

NETWORK
TITLE =controllers

      NOP   0;
// CO2BRV1 PID 001 CO2 B RV1
      CALL FC    55 (
           UnitNo                   := #UnitNo,
           PIDRec                   := DB2266.CO2BRV1,
           SpExt                    := DB2266.DBD  234,
           PVal                     := DB2266.DBD  254,
           OPer                     := PQW  222);

NETWORK
TITLE =unit supply

      UC    FB [#UnitFB];

NETWORK
TITLE =B_G1  B_G1
// Act 001
// Box           : VS2-BB
// Output address: Q309.4
      CALL FC    70 (
           UnitNo                   := #UnitNo,
           ActRec                   := DB2260.B_G1,
           Typ                      := 1,
           FBa                      := #xTmp,
           FBa2                     := I    309.4,
           Out                      := Q    309.4);

NETWORK
TITLE =CO2_BV2  Ansteuerung BV2
// Act 002
// Box           : CO2 Dosierung
// Output address: Q61.6
      CALL FC    70 (
           UnitNo                   := #UnitNo,
           ActRec                   := DB2260.CO2_BV2,
           Typ                      := 0,
           FBa                      := #xTmp,
           FBa2                     := #xTmp,
           Out                      := Q     61.6);

NETWORK
TITLE =CO2_BV1  Ansteuerung BV1
// Act 003
// Box           : CO2 Dosierung
// Output address: Q60.6
      CALL FC    70 (
           UnitNo                   := #UnitNo,
           ActRec                   := DB2260.CO2_BV1,
           Typ                      := 0,
           FBa                      := #xTmp,
           FBa2                     := #xTmp,
           Out                      := Q     60.6);

NETWORK
TITLE =BRV1  CO2 B RV1
// Act 004
// Box           :
// Input address : #xtmp
// Output address: #xtmp
      CALL FC    70 (
           UnitNo                   := #UnitNo,
           ActRec                   := DB2260.BRV1,
           Typ                      := 4,
           FBa                      := #xTmp,
           FBa2                     := #xTmp,
           Out                      := #xTmp);

END_FUNCTION_BLOCK

FUNCTION_BLOCK FB 1261
TITLE =U026: Well Transfer B
FAMILY : BOTEC_F1
NAME : UniE
VERSION : 1.2


VAR_TEMP
  CIP : BOOL ;	//CIP active
  UNIM : BOOL ;	//Unit Not In Maintenance
  GenRel : BOOL ;	//general OK (emergency and maintenance OK)
  EStopOK : BOOL ;	//emergency OK
  UnitNo : INT ;	//unit number
  xTmp : BOOL ;	//Temporary Bool
  iTmp : INT ;	//Temporary INT
  rTmp : REAL ;	//Temporary REAL
  dTmp : DINT ;	//Temporary DINT (free for general use)
  RetValInt : INT ;	//return value
END_VAR
BEGIN
NETWORK
TITLE =General

      SET   ;
// Simulation ---------------------------------------------------------------
      A     DB1261.DBX 1357.7;
      CC    FB  1269; // "U026Sim"
      A     DB1261.DBX   17.3;
      =     DB1261.DBX 1357.7; //Help bit for simulation

// get unit number ----------------------------------------------------------
      L     DB1260.DBW    0;
      T     #UnitNo;

// communication ------------------------------------------------------------
      UC    FB  1265; // U026Com

NETWORK
TITLE =Sequence organisation

      CLR   ;
      =     M    122.2;

// sequencer ----------------------------------------------------------------
      A     DB1263.DBX   43.1;
      S     DB1263.DBX   97.3;

      CALL FC    40 (
           UnitNo                   := #UnitNo);

END_FUNCTION_BLOCK

FUNCTION_BLOCK FB 1270
TITLE =U027: Well Transfer CF
FAMILY : BOTEC_F1
NAME : UniA
VERSION : 2.1


VAR_TEMP
  EStopOK : BOOL ;	//auxiliary flag
  CIP : BOOL ;	//CIP Program Selected
  xTmp : BOOL ;	//Temporary Bool(free for general use)
  UnitNo : INT ;	//unit number
  UnitFB : INT ;	//unit expansion FB number
  rTmp : REAL ;	//Temporary REAL (free for general use)
  iTmp : INT ;	//Temporary INT (free for general use)
  dTmp : DINT ;	//Temporary DINT (free for general use)
END_VAR
BEGIN
NETWORK
TITLE =general

      CLR   ;
      =     #xTmp;
      =     #EStopOK;

      L     DB1270.DBW    0;
      T     #UnitNo;
      L     DB1270.DBW    2;
      T     #UnitFB;

NETWORK
TITLE =analog inputs

      NOP   0;
// C_AnI01 AnI 001 spare
      CALL FC    24 (
           UnitNo                   := #UnitNo,
           AnIRec                   := DB2273.C_AnI01,
           ValPer                   := #iTmp);

// QI_CO2_CF_PH AnI 002
      CALL FC    24 (
           UnitNo                   := #UnitNo,
           AnIRec                   := DB2273.QI_CO2_CF_PH,
           ValPer                   := IW   550);

// AnI03 AnI 003 spare
      CALL FC    24 (
           UnitNo                   := #UnitNo,
           AnIRec                   := DB2273.AnI03,
           ValPer                   := #iTmp);

NETWORK
TITLE =Universal value

      NOP   0;
// unv001 UnV 001 Process Status
      CALL FC    27 (
           UnitNo                   := #UnitNo,
           UnVRec                   := DB2275.unv001,
           ValExt                   := DB2275.DBD  234);

// unv002 UnV 002 Universal Value 02
      CALL FC    27 (
           UnitNo                   := #UnitNo,
           UnVRec                   := DB2275.unv002,
           ValExt                   := DB2275.DBD  362);

// unv003 UnV 003 Universal Value 03
      CALL FC    27 (
           UnitNo                   := #UnitNo,
           UnVRec                   := DB2275.unv003,
           ValExt                   := DB2275.DBD  490);

// unv004 UnV 004 Universal Value 04
      CALL FC    27 (
           UnitNo                   := #UnitNo,
           UnVRec                   := DB2275.unv004,
           ValExt                   := DB2275.DBD  618);

NETWORK
TITLE =special inputs

      NOP   0;
// SpI01 SpI 001 spare
      CALL FC    14 (
           UnitNo                   := #UnitNo,
           SpIRec                   := DB2271.SpI01,
           SpIBit                   := #xTmp);

// SpI02 SpI 002 spare
      CALL FC    14 (
           UnitNo                   := #UnitNo,
           SpIRec                   := DB2271.SpI02,
           SpIBit                   := #xTmp);

// SpI03 SpI 003 spare
      CALL FC    14 (
           UnitNo                   := #UnitNo,
           SpIRec                   := DB2271.SpI03,
           SpIBit                   := #xTmp);

// SpI04 SpI 004 spare
      CALL FC    14 (
           UnitNo                   := #UnitNo,
           SpIRec                   := DB2271.SpI04,
           SpIBit                   := #xTmp);

NETWORK
TITLE =messages

      NOP   0;
// msg001 Msg 001 Message 01
      CALL FC    16 (
           UnitNo                   := #UnitNo,
           MsgRec                   := DB2277.msg001,
           MsgBit                   := DB2277.DBX   82.7);

// msg002 Msg 002 Message 02
      CALL FC    16 (
           UnitNo                   := #UnitNo,
           MsgRec                   := DB2277.msg002,
           MsgBit                   := DB2277.DBX  142.7);

// msg003 Msg 003 Message 03
      CALL FC    16 (
           UnitNo                   := #UnitNo,
           MsgRec                   := DB2277.msg003,
           MsgBit                   := DB2277.DBX  202.7);

NETWORK
TITLE =controllers

      NOP   0;
// CO2CFRV1 PID 001 CO2 CF RV1
      CALL FC    55 (
           UnitNo                   := #UnitNo,
           PIDRec                   := DB2276.CO2CFRV1,
           SpExt                    := DB2276.DBD  234,
           PVal                     := DB2276.DBD  254,
           OPer                     := PQW  550);

NETWORK
TITLE =unit supply

      UC    FB [#UnitFB];

NETWORK
TITLE =CF_G1
// Act 001
// Box           : Ventilinsel 1
// Input address : I16.5
// Output address: Q16.5
      CALL FC    70 (
           UnitNo                   := #UnitNo,
           ActRec                   := DB2270.CF_G1,
           Typ                      := 1,
           FBa                      := #xTmp,
           FBa2                     := I     16.5,
           Out                      := Q     16.5);

NETWORK
TITLE =CO2_CFV2
// Act 002
// Box           : CO2 Dosierung
// Output address: Q62.3
      CALL FC    70 (
           UnitNo                   := #UnitNo,
           ActRec                   := DB2270.CO2_CFV2,
           Typ                      := 0,
           FBa                      := #xTmp,
           FBa2                     := #xTmp,
           Out                      := Q     62.3);

NETWORK
TITLE =CO2_CFV1
// Act 003
// Box           : CO2 Dosierung
// Output address: Q62.2
      CALL FC    70 (
           UnitNo                   := #UnitNo,
           ActRec                   := DB2270.CO2_CFV1,
           Typ                      := 0,
           FBa                      := #xTmp,
           FBa2                     := #xTmp,
           Out                      := Q     62.2);

NETWORK
TITLE =CFRV1  CO2 CF RV1
// Act 004
// Box           :
// Output address: #xtmp
      CALL FC    70 (
           UnitNo                   := #UnitNo,
           ActRec                   := DB2270.CFRV1,
           Typ                      := 0,
           FBa                      := #xTmp,
           FBa2                     := #xTmp,
           Out                      := #xTmp);

END_FUNCTION_BLOCK

FUNCTION_BLOCK FB 1271
TITLE =U027: Well Transfer CF
FAMILY : BOTEC_F1
NAME : UniE
VERSION : 1.2


VAR_TEMP
  CIP : BOOL ;	//CIP active
  UNIM : BOOL ;	//Unit Not In Maintenance
  GenRel : BOOL ;	//general OK (emergency and maintenance OK)
  EStopOK : BOOL ;	//emergency OK
  UnitNo : INT ;	//unit number
  xTmp : BOOL ;	//Temporary Bool
  iTmp : INT ;	//Temporary INT
  rTmp : REAL ;	//Temporary REAL
  dTmp : DINT ;	//Temporary DINT (free for general use)
  RetValInt : INT ;	//return value
END_VAR
BEGIN
NETWORK
TITLE =General

      SET   ;
// Simulation ---------------------------------------------------------------
      A     DB1271.DBX 1357.7;
      CC    FB  1279; // "U027Sim"
      A     DB1271.DBX   17.3;
      =     DB1271.DBX 1357.7; //Help bit for simulation

// get unit number ----------------------------------------------------------
      L     DB1270.DBW    0;
      T     #UnitNo;

// communication ------------------------------------------------------------
      UC    FB  1275; // U027Com

NETWORK
TITLE =Sequence organisation

      CLR   ;
      =     M    122.2;

// sequencer ----------------------------------------------------------------
      A     DB1273.DBX   43.1;
      S     DB1273.DBX   97.3;

      CALL FC    40 (
           UnitNo                   := #UnitNo);

END_FUNCTION_BLOCK

FUNCTION_BLOCK FB 1280
TITLE =U028: Well Transfer C
FAMILY : BOTEC_F1
NAME : UniA
VERSION : 2.1


VAR_TEMP
  EStopOK : BOOL ;	//auxiliary flag
  CIP : BOOL ;	//CIP Program Selected
  xTmp : BOOL ;	//Temporary Bool(free for general use)
  UnitNo : INT ;	//unit number
  UnitFB : INT ;	//unit expansion FB number
  rTmp : REAL ;	//Temporary REAL (free for general use)
  iTmp : INT ;	//Temporary INT (free for general use)
  dTmp : DINT ;	//Temporary DINT (free for general use)
END_VAR
BEGIN
NETWORK
TITLE =general

      CLR   ;
      =     #xTmp;
      =     #EStopOK;

      L     DB1280.DBW    0;
      T     #UnitNo;
      L     DB1280.DBW    2;
      T     #UnitFB;

NETWORK
TITLE =analog inputs

      NOP   0;
// C_AnI01 AnI 001 spare
      CALL FC    24 (
           UnitNo                   := #UnitNo,
           AnIRec                   := DB2283.C_AnI01,
           ValPer                   := #iTmp);

// QI_CO2_C_PH AnI 002
      CALL FC    24 (
           UnitNo                   := #UnitNo,
           AnIRec                   := DB2283.QI_CO2_C_PH,
           ValPer                   := IW   548);

// AnI03 AnI 003 spare
      CALL FC    24 (
           UnitNo                   := #UnitNo,
           AnIRec                   := DB2283.AnI03,
           ValPer                   := #iTmp);

NETWORK
TITLE =Universal value

      NOP   0;
// unv001 UnV 001 Process Status
      CALL FC    27 (
           UnitNo                   := #UnitNo,
           UnVRec                   := DB2285.unv001,
           ValExt                   := DB2285.DBD  234);

// unv002 UnV 002 Universal Value 02
      CALL FC    27 (
           UnitNo                   := #UnitNo,
           UnVRec                   := DB2285.unv002,
           ValExt                   := DB2285.DBD  362);

// unv003 UnV 003 Universal Value 03
      CALL FC    27 (
           UnitNo                   := #UnitNo,
           UnVRec                   := DB2285.unv003,
           ValExt                   := DB2285.DBD  490);

// unv004 UnV 004 Universal Value 04
      CALL FC    27 (
           UnitNo                   := #UnitNo,
           UnVRec                   := DB2285.unv004,
           ValExt                   := DB2285.DBD  618);

NETWORK
TITLE =special inputs

      NOP   0;
// SpI01 SpI 001 spare
      CALL FC    14 (
           UnitNo                   := #UnitNo,
           SpIRec                   := DB2281.SpI01,
           SpIBit                   := #xTmp);

// SpI02 SpI 002 spare
      CALL FC    14 (
           UnitNo                   := #UnitNo,
           SpIRec                   := DB2281.SpI02,
           SpIBit                   := #xTmp);

// SpI03 SpI 003 spare
      CALL FC    14 (
           UnitNo                   := #UnitNo,
           SpIRec                   := DB2281.SpI03,
           SpIBit                   := #xTmp);

// SpI04 SpI 004 spare
      CALL FC    14 (
           UnitNo                   := #UnitNo,
           SpIRec                   := DB2281.SpI04,
           SpIBit                   := #xTmp);

NETWORK
TITLE =messages

      NOP   0;
// msg001 Msg 001 Message 01
      CALL FC    16 (
           UnitNo                   := #UnitNo,
           MsgRec                   := DB2287.msg001,
           MsgBit                   := DB2287.DBX   82.7);

// msg002 Msg 002 Message 02
      CALL FC    16 (
           UnitNo                   := #UnitNo,
           MsgRec                   := DB2287.msg002,
           MsgBit                   := DB2287.DBX  142.7);

// msg003 Msg 003 Message 03
      CALL FC    16 (
           UnitNo                   := #UnitNo,
           MsgRec                   := DB2287.msg003,
           MsgBit                   := DB2287.DBX  202.7);

NETWORK
TITLE =controllers

      NOP   0;
// CO2CRV1 PID 001 CO2 C RV1
      CALL FC    55 (
           UnitNo                   := #UnitNo,
           PIDRec                   := DB2286.CO2CRV1,
           SpExt                    := DB2286.DBD  234,
           PVal                     := DB2286.DBD  254,
           OPer                     := PQW  548);

NETWORK
TITLE =unit supply

      UC    FB [#UnitFB];

NETWORK
TITLE =C_G1
// Act 001
// Box           : Ventilinsel 1
// Input address : I17.7
// Output address: Q17.7
      CALL FC    70 (
           UnitNo                   := #UnitNo,
           ActRec                   := DB2280.C_G1,
           Typ                      := 1,
           FBa                      := #xTmp,
           FBa2                     := I     17.7,
           Out                      := Q     17.7);

NETWORK
TITLE =CO2_CV2
// Act 002
// Box           : CO2 Dosierung
// Output address: Q62.1
      CALL FC    70 (
           UnitNo                   := #UnitNo,
           ActRec                   := DB2280.CO2_CV2,
           Typ                      := 0,
           FBa                      := #xTmp,
           FBa2                     := #xTmp,
           Out                      := Q     62.1);

NETWORK
TITLE =CO2_CV1
// Act 003
// Box           : CO2 Dosierung
// Output address: Q62.0
      CALL FC    70 (
           UnitNo                   := #UnitNo,
           ActRec                   := DB2280.CO2_CV1,
           Typ                      := 0,
           FBa                      := #xTmp,
           FBa2                     := #xTmp,
           Out                      := Q     62.0);

NETWORK
TITLE =CRV1  CO2 C RV1
// Act 004
// Box           :
// Input address : #xtmp
// Output address: #xtmp
      CALL FC    70 (
           UnitNo                   := #UnitNo,
           ActRec                   := DB2280.CRV1,
           Typ                      := 4,
           FBa                      := #xTmp,
           FBa2                     := #xTmp,
           Out                      := #xTmp);

END_FUNCTION_BLOCK

FUNCTION_BLOCK FB 1281
TITLE =U028: Well Transfer C
FAMILY : BOTEC_F1
NAME : UniE
VERSION : 1.2


VAR_TEMP
  CIP : BOOL ;	//CIP active
  UNIM : BOOL ;	//Unit Not In Maintenance
  GenRel : BOOL ;	//general OK (emergency and maintenance OK)
  EStopOK : BOOL ;	//emergency OK
  UnitNo : INT ;	//unit number
  xTmp : BOOL ;	//Temporary Bool
  iTmp : INT ;	//Temporary INT
  rTmp : REAL ;	//Temporary REAL
  dTmp : DINT ;	//Temporary DINT (free for general use)
  RetValInt : INT ;	//return value
END_VAR
BEGIN
NETWORK
TITLE =General

      SET   ;
// Simulation ---------------------------------------------------------------
      A     DB1281.DBX 1357.7;
      CC    FB  1289; // "U028Sim"
      A     DB1281.DBX   17.3;
      =     DB1281.DBX 1357.7; //Help bit for simulation

// get unit number ----------------------------------------------------------
      L     DB1280.DBW    0;
      T     #UnitNo;

// communication ------------------------------------------------------------
      UC    FB  1285; // U028Com

NETWORK
TITLE =Sequence organisation

      CLR   ;
      =     M    122.2;

// sequencer ----------------------------------------------------------------
      A     DB1283.DBX   43.1;
      S     DB1283.DBX   97.3;

      CALL FC    40 (
           UnitNo                   := #UnitNo);

END_FUNCTION_BLOCK

FUNCTION_BLOCK FB 1290
TITLE =U029: Well Transfer B6F
FAMILY : BOTEC_F1
NAME : UniA
VERSION : 2.1


VAR_TEMP
  EStopOK : BOOL ;	//auxiliary flag
  CIP : BOOL ;	//CIP Program Selected
  xTmp : BOOL ;	//Temporary Bool(free for general use)
  UnitNo : INT ;	//unit number
  UnitFB : INT ;	//unit expansion FB number
  rTmp : REAL ;	//Temporary REAL (free for general use)
  iTmp : INT ;	//Temporary INT (free for general use)
  dTmp : DINT ;	//Temporary DINT (free for general use)
END_VAR
BEGIN
NETWORK
TITLE =general

      CLR   ;
      =     #xTmp;
      =     #EStopOK;

      L     DB1290.DBW    0;
      T     #UnitNo;
      L     DB1290.DBW    2;
      T     #UnitFB;

NETWORK
TITLE =analog inputs

      NOP   0;
// C_AnI01 AnI 001 spare
      CALL FC    24 (
           UnitNo                   := #UnitNo,
           AnIRec                   := DB2293.C_AnI01,
           ValPer                   := #iTmp);

// QI_CO2_B6F_PH AnI 002
      CALL FC    24 (
           UnitNo                   := #UnitNo,
           AnIRec                   := DB2293.QI_CO2_B6F_PH,
           ValPer                   := IW   216);

// AnI03 AnI 003 spare
      CALL FC    24 (
           UnitNo                   := #UnitNo,
           AnIRec                   := DB2293.AnI03,
           ValPer                   := #iTmp);

NETWORK
TITLE =Universal value

      NOP   0;
// unv001 UnV 001 Process Status
      CALL FC    27 (
           UnitNo                   := #UnitNo,
           UnVRec                   := DB2295.unv001,
           ValExt                   := DB2295.DBD  234);

// unv002 UnV 002 Universal Value 02
      CALL FC    27 (
           UnitNo                   := #UnitNo,
           UnVRec                   := DB2295.unv002,
           ValExt                   := DB2295.DBD  362);

// unv003 UnV 003 Universal Value 03
      CALL FC    27 (
           UnitNo                   := #UnitNo,
           UnVRec                   := DB2295.unv003,
           ValExt                   := DB2295.DBD  490);

// unv004 UnV 004 Universal Value 04
      CALL FC    27 (
           UnitNo                   := #UnitNo,
           UnVRec                   := DB2295.unv004,
           ValExt                   := DB2295.DBD  618);

NETWORK
TITLE =special inputs

      NOP   0;
// RM_NI_KF2_K1 SpI 001 PANEEL PTV1
      CALL FC    14 (
           UnitNo                   := #UnitNo,
           SpIRec                   := DB2291.RM_NI_KF2_K1,
           SpIBit                   := I     54.7);

// RM_NI_KF2_K2 SpI 002 PANEEL PTV1
      CALL FC    14 (
           UnitNo                   := #UnitNo,
           SpIRec                   := DB2291.RM_NI_KF2_K2,
           SpIBit                   := I     55.0);

// RM_NI_KF2_K3 SpI 003 PANEEL PTV1
      CALL FC    14 (
           UnitNo                   := #UnitNo,
           SpIRec                   := DB2291.RM_NI_KF2_K3,
           SpIBit                   := I     55.1);

// SpI04 SpI 004 spare
      CALL FC    14 (
           UnitNo                   := #UnitNo,
           SpIRec                   := DB2291.SpI04,
           SpIBit                   := #xTmp);

NETWORK
TITLE =messages

      NOP   0;
// msg001 Msg 001 Message 01
      CALL FC    16 (
           UnitNo                   := #UnitNo,
           MsgRec                   := DB2297.msg001,
           MsgBit                   := DB2297.DBX   82.7);

// msg002 Msg 002 Message 02
      CALL FC    16 (
           UnitNo                   := #UnitNo,
           MsgRec                   := DB2297.msg002,
           MsgBit                   := DB2297.DBX  142.7);

// msg003 Msg 003 Message 03
      CALL FC    16 (
           UnitNo                   := #UnitNo,
           MsgRec                   := DB2297.msg003,
           MsgBit                   := DB2297.DBX  202.7);

NETWORK
TITLE =controllers

      NOP   0;
// CO2B6FRV1 PID 001 CO2 B6F RV1
      CALL FC    55 (
           UnitNo                   := #UnitNo,
           PIDRec                   := DB2296.CO2B6FRV1,
           SpExt                    := DB2296.DBD  234,
           PVal                     := DB2296.DBD  254,
           OPer                     := PQW  216);

NETWORK
TITLE =unit supply

      UC    FB [#UnitFB];

NETWORK
TITLE =B6F_G1  B6F_G1
// Act 001
// Box           : VS2-BB
// Output address: Q309.6
      CALL FC    70 (
           UnitNo                   := #UnitNo,
           ActRec                   := DB2290.B6F_G1,
           Typ                      := 1,
           FBa                      := #xTmp,
           FBa2                     := I    309.6,
           Out                      := Q    309.6);

NETWORK
TITLE =CO2_B6FV2  Ansteuerung B6FV2
// Act 002
// Box           : CO2 Dosierung
// Output address: Q61.0
      CALL FC    70 (
           UnitNo                   := #UnitNo,
           ActRec                   := DB2290.CO2_B6FV2,
           Typ                      := 0,
           FBa                      := #xTmp,
           FBa2                     := #xTmp,
           Out                      := Q     61.0);

NETWORK
TITLE =CO2_B6FV1  Ansteuerung B6FV1
// Act 003
// Box           : CO2 Dosierung
// Output address: Q60.0
      CALL FC    70 (
           UnitNo                   := #UnitNo,
           ActRec                   := DB2290.CO2_B6FV1,
           Typ                      := 0,
           FBa                      := #xTmp,
           FBa2                     := #xTmp,
           Out                      := Q     60.0);

NETWORK
TITLE =B6FRV1  CO2 B6F RV1
// Act 004
// Box           :
// Input address : #xtmp
// Output address: #xtmp
      CALL FC    70 (
           UnitNo                   := #UnitNo,
           ActRec                   := DB2290.B6FRV1,
           Typ                      := 4,
           FBa                      := #xTmp,
           FBa2                     := #xTmp,
           Out                      := #xTmp);

END_FUNCTION_BLOCK

FUNCTION_BLOCK FB 1291
TITLE =U029: Well Transfer B6F
FAMILY : BOTEC_F1
NAME : UniE
VERSION : 1.2


VAR_TEMP
  CIP : BOOL ;	//CIP active
  UNIM : BOOL ;	//Unit Not In Maintenance
  GenRel : BOOL ;	//general OK (emergency and maintenance OK)
  EStopOK : BOOL ;	//emergency OK
  UnitNo : INT ;	//unit number
  xTmp : BOOL ;	//Temporary Bool
  iTmp : INT ;	//Temporary INT
  rTmp : REAL ;	//Temporary REAL
  dTmp : DINT ;	//Temporary DINT (free for general use)
  RetValInt : INT ;	//return value
END_VAR
BEGIN
NETWORK
TITLE =General

      SET   ;
// Simulation ---------------------------------------------------------------
      A     DB1291.DBX 1357.7;
      CC    FB  1299; // "U029Sim"
      A     DB1291.DBX   17.3;
      =     DB1291.DBX 1357.7; //Help bit for simulation

// get unit number ----------------------------------------------------------
      L     DB1290.DBW    0;
      T     #UnitNo;

// communication ------------------------------------------------------------
      UC    FB  1295; // U029Com

NETWORK
TITLE =Sequence organisation

      CLR   ;
      =     M    122.2;

// sequencer ----------------------------------------------------------------
      A     DB1293.DBX   43.1;
      S     DB1293.DBX   97.3;

      CALL FC    40 (
           UnitNo                   := #UnitNo);

END_FUNCTION_BLOCK

FUNCTION_BLOCK FB 1300
TITLE =U030: Well Transfer H6
FAMILY : BOTEC_F1
NAME : UniA
VERSION : 2.1


VAR_TEMP
  EStopOK : BOOL ;	//auxiliary flag
  CIP : BOOL ;	//CIP Program Selected
  xTmp : BOOL ;	//Temporary Bool(free for general use)
  UnitNo : INT ;	//unit number
  UnitFB : INT ;	//unit expansion FB number
  rTmp : REAL ;	//Temporary REAL (free for general use)
  iTmp : INT ;	//Temporary INT (free for general use)
  dTmp : DINT ;	//Temporary DINT (free for general use)
END_VAR
BEGIN
NETWORK
TITLE =general

      CLR   ;
      =     #xTmp;
      =     #EStopOK;

      L     DB1300.DBW    0;
      T     #UnitNo;
      L     DB1300.DBW    2;
      T     #UnitFB;

NETWORK
TITLE =analog inputs

      NOP   0;
// C_AnI01 AnI 001 spare
      CALL FC    24 (
           UnitNo                   := #UnitNo,
           AnIRec                   := DB2303.C_AnI01,
           ValPer                   := #iTmp);

// QI_CO2_H6F_PH AnI 002
      CALL FC    24 (
           UnitNo                   := #UnitNo,
           AnIRec                   := DB2303.QI_CO2_H6F_PH,
           ValPer                   := IW   218);

// AnI03 AnI 003 spare
      CALL FC    24 (
           UnitNo                   := #UnitNo,
           AnIRec                   := DB2303.AnI03,
           ValPer                   := #iTmp);

NETWORK
TITLE =Universal value

      NOP   0;
// unv001 UnV 001 Process Status
      CALL FC    27 (
           UnitNo                   := #UnitNo,
           UnVRec                   := DB2305.unv001,
           ValExt                   := DB2305.DBD  234);

// unv002 UnV 002 Universal Value 02
      CALL FC    27 (
           UnitNo                   := #UnitNo,
           UnVRec                   := DB2305.unv002,
           ValExt                   := DB2305.DBD  362);

// unv003 UnV 003 Universal Value 03
      CALL FC    27 (
           UnitNo                   := #UnitNo,
           UnVRec                   := DB2305.unv003,
           ValExt                   := DB2305.DBD  490);

// unv004 UnV 004 Universal Value 04
      CALL FC    27 (
           UnitNo                   := #UnitNo,
           UnVRec                   := DB2305.unv004,
           ValExt                   := DB2305.DBD  618);

NETWORK
TITLE =special inputs

      NOP   0;
// SpI01 SpI 001 spare
      CALL FC    14 (
           UnitNo                   := #UnitNo,
           SpIRec                   := DB2301.SpI01,
           SpIBit                   := #xTmp);

// SpI02 SpI 002 spare
      CALL FC    14 (
           UnitNo                   := #UnitNo,
           SpIRec                   := DB2301.SpI02,
           SpIBit                   := #xTmp);

// SpI03 SpI 003 spare
      CALL FC    14 (
           UnitNo                   := #UnitNo,
           SpIRec                   := DB2301.SpI03,
           SpIBit                   := #xTmp);

// SpI04 SpI 004 spare
      CALL FC    14 (
           UnitNo                   := #UnitNo,
           SpIRec                   := DB2301.SpI04,
           SpIBit                   := #xTmp);

NETWORK
TITLE =messages

      NOP   0;
// msg001 Msg 001 Message 01
      CALL FC    16 (
           UnitNo                   := #UnitNo,
           MsgRec                   := DB2307.msg001,
           MsgBit                   := DB2307.DBX   82.7);

// msg002 Msg 002 Message 02
      CALL FC    16 (
           UnitNo                   := #UnitNo,
           MsgRec                   := DB2307.msg002,
           MsgBit                   := DB2307.DBX  142.7);

// msg003 Msg 003 Message 03
      CALL FC    16 (
           UnitNo                   := #UnitNo,
           MsgRec                   := DB2307.msg003,
           MsgBit                   := DB2307.DBX  202.7);

NETWORK
TITLE =controllers

      NOP   0;
// CO2H6FRV1 PID 001 CO2 H6F RV1
      CALL FC    55 (
           UnitNo                   := #UnitNo,
           PIDRec                   := DB2306.CO2H6FRV1,
           SpExt                    := DB2306.DBD  234,
           PVal                     := DB2306.DBD  254,
           OPer                     := PQW  218);

NETWORK
TITLE =unit supply

      UC    FB [#UnitFB];

NETWORK
TITLE =H6F_G1  H6F_G1
// Act 001
// Box           : VS2-BB
// Output address: Q309.5
      CALL FC    70 (
           UnitNo                   := #UnitNo,
           ActRec                   := DB2300.H6F_G1,
           Typ                      := 1,
           FBa                      := #xTmp,
           FBa2                     := I    309.5,
           Out                      := Q    309.5);

NETWORK
TITLE =CO2_H6FV2  Ansteuerung H6FV2
// Act 002
// Box           : CO2 Dosierung
// Output address: Q61.1
      CALL FC    70 (
           UnitNo                   := #UnitNo,
           ActRec                   := DB2300.CO2_H6FV2,
           Typ                      := 0,
           FBa                      := #xTmp,
           FBa2                     := #xTmp,
           Out                      := Q     61.1);

NETWORK
TITLE =CO2_H6FV1  Ansteuerung H6FV1
// Act 003
// Box           : CO2 Dosierung
// Output address: Q60.1
      CALL FC    70 (
           UnitNo                   := #UnitNo,
           ActRec                   := DB2300.CO2_H6FV1,
           Typ                      := 0,
           FBa                      := #xTmp,
           FBa2                     := #xTmp,
           Out                      := Q     60.1);

NETWORK
TITLE =H6RV1  CO2 H6 RV1
// Act 004
// Box           :
// Input address : #xtmp
// Output address: #xtmp
      CALL FC    70 (
           UnitNo                   := #UnitNo,
           ActRec                   := DB2300.H6RV1,
           Typ                      := 4,
           FBa                      := #xTmp,
           FBa2                     := #xTmp,
           Out                      := #xTmp);

END_FUNCTION_BLOCK

FUNCTION_BLOCK FB 1301
TITLE =U030: Well Transfer H6
FAMILY : BOTEC_F1
NAME : UniE
VERSION : 1.2


VAR_TEMP
  CIP : BOOL ;	//CIP active
  UNIM : BOOL ;	//Unit Not In Maintenance
  GenRel : BOOL ;	//general OK (emergency and maintenance OK)
  EStopOK : BOOL ;	//emergency OK
  UnitNo : INT ;	//unit number
  xTmp : BOOL ;	//Temporary Bool
  iTmp : INT ;	//Temporary INT
  rTmp : REAL ;	//Temporary REAL
  dTmp : DINT ;	//Temporary DINT (free for general use)
  RetValInt : INT ;	//return value
END_VAR
BEGIN
NETWORK
TITLE =General

      SET   ;
// Simulation ---------------------------------------------------------------
      A     DB1301.DBX 1357.7;
      CC    FB  1309; // "U030Sim"
      A     DB1301.DBX   17.3;
      =     DB1301.DBX 1357.7; //Help bit for simulation

// get unit number ----------------------------------------------------------
      L     DB1300.DBW    0;
      T     #UnitNo;

// communication ------------------------------------------------------------
      UC    FB  1305; // U030Com

NETWORK
TITLE =Sequence organisation

      CLR   ;
      =     M    122.2;

// sequencer ----------------------------------------------------------------
      A     DB1303.DBX   43.1;
      S     DB1303.DBX   97.3;

      CALL FC    40 (
           UnitNo                   := #UnitNo);

END_FUNCTION_BLOCK

FUNCTION_BLOCK FB 1310
TITLE =U031: Well Transfer J6
FAMILY : BOTEC_F1
NAME : UniA
VERSION : 2.1


VAR_TEMP
  EStopOK : BOOL ;	//auxiliary flag
  CIP : BOOL ;	//CIP Program Selected
  xTmp : BOOL ;	//Temporary Bool(free for general use)
  UnitNo : INT ;	//unit number
  UnitFB : INT ;	//unit expansion FB number
  rTmp : REAL ;	//Temporary REAL (free for general use)
  iTmp : INT ;	//Temporary INT (free for general use)
  dTmp : DINT ;	//Temporary DINT (free for general use)
END_VAR
BEGIN
NETWORK
TITLE =general

      CLR   ;
      =     #xTmp;
      =     #EStopOK;

      L     DB1310.DBW    0;
      T     #UnitNo;
      L     DB1310.DBW    2;
      T     #UnitFB;

NETWORK
TITLE =analog inputs

      NOP   0;
// J6F_Druck AnI 001 J6F_Druck
      CALL FC    24 (
           UnitNo                   := #UnitNo,
           AnIRec                   := DB2313.J6F_Druck,
           ValPer                   := #iTmp);

// QI_CO2_J6F_PH AnI 002
      CALL FC    24 (
           UnitNo                   := #UnitNo,
           AnIRec                   := DB2313.QI_CO2_J6F_PH,
           ValPer                   := IW   208);

// AnI03 AnI 003 spare
      CALL FC    24 (
           UnitNo                   := #UnitNo,
           AnIRec                   := DB2313.AnI03,
           ValPer                   := #iTmp);

NETWORK
TITLE =Universal value

      NOP   0;
// unv001 UnV 001 Process Status
      CALL FC    27 (
           UnitNo                   := #UnitNo,
           UnVRec                   := DB2315.unv001,
           ValExt                   := DB2315.DBD  234);

// unv002 UnV 002 Universal Value 02
      CALL FC    27 (
           UnitNo                   := #UnitNo,
           UnVRec                   := DB2315.unv002,
           ValExt                   := DB2315.DBD  362);

// unv003 UnV 003 Universal Value 03
      CALL FC    27 (
           UnitNo                   := #UnitNo,
           UnVRec                   := DB2315.unv003,
           ValExt                   := DB2315.DBD  490);

// unv004 UnV 004 Universal Value 04
      CALL FC    27 (
           UnitNo                   := #UnitNo,
           UnVRec                   := DB2315.unv004,
           ValExt                   := DB2315.DBD  618);

NETWORK
TITLE =special inputs

      NOP   0;
// SpI01 SpI 001 spare
      CALL FC    14 (
           UnitNo                   := #UnitNo,
           SpIRec                   := DB2311.SpI01,
           SpIBit                   := #xTmp);

// SpI02 SpI 002 spare
      CALL FC    14 (
           UnitNo                   := #UnitNo,
           SpIRec                   := DB2311.SpI02,
           SpIBit                   := #xTmp);

// SpI03 SpI 003 spare
      CALL FC    14 (
           UnitNo                   := #UnitNo,
           SpIRec                   := DB2311.SpI03,
           SpIBit                   := #xTmp);

// SpI04 SpI 004 spare
      CALL FC    14 (
           UnitNo                   := #UnitNo,
           SpIRec                   := DB2311.SpI04,
           SpIBit                   := #xTmp);

NETWORK
TITLE =messages

      NOP   0;
// msg001 Msg 001 Message 01
      CALL FC    16 (
           UnitNo                   := #UnitNo,
           MsgRec                   := DB2317.msg001,
           MsgBit                   := DB2317.DBX   82.7);

// msg002 Msg 002 Message 02
      CALL FC    16 (
           UnitNo                   := #UnitNo,
           MsgRec                   := DB2317.msg002,
           MsgBit                   := DB2317.DBX  142.7);

// msg003 Msg 003 Message 03
      CALL FC    16 (
           UnitNo                   := #UnitNo,
           MsgRec                   := DB2317.msg003,
           MsgBit                   := DB2317.DBX  202.7);

NETWORK
TITLE =controllers

      NOP   0;
// CO2J6FRV1 PID 001 CO2 J6F RV1
      CALL FC    55 (
           UnitNo                   := #UnitNo,
           PIDRec                   := DB2316.CO2J6FRV1,
           SpExt                    := DB2316.DBD  234,
           PVal                     := DB2316.DBD  254,
           OPer                     := PQW  540);

NETWORK
TITLE =unit supply

      UC    FB [#UnitFB];

NETWORK
TITLE =J6F_G1  J6F_G1
// Act 001
// Box           : VS2-BB
// Output address: Q309.7
      CALL FC    70 (
           UnitNo                   := #UnitNo,
           ActRec                   := DB2310.J6F_G1,
           Typ                      := 1,
           FBa                      := #xTmp,
           FBa2                     := I    309.7,
           Out                      := Q    309.7);

NETWORK
TITLE =CO2_J6FV2  Ansteuerung J6FV2
// Act 002
// Box           : CO2 Dosierung
// Output address: Q61.2
      CALL FC    70 (
           UnitNo                   := #UnitNo,
           ActRec                   := DB2310.CO2_J6FV2,
           Typ                      := 0,
           FBa                      := #xTmp,
           FBa2                     := #xTmp,
           Out                      := Q     61.2);

NETWORK
TITLE =CO2_J6FV1  Ansteuerung J6FV1
// Act 003
// Box           : CO2 Dosierung
// Output address: Q60.2
      CALL FC    70 (
           UnitNo                   := #UnitNo,
           ActRec                   := DB2310.CO2_J6FV1,
           Typ                      := 0,
           FBa                      := #xTmp,
           FBa2                     := #xTmp,
           Out                      := Q     60.2);

NETWORK
TITLE =J6FRV1  CO2 J6F RV1
// Act 004
// Box           :
// Input address : #xtmp
// Output address: #xtmp
      CALL FC    70 (
           UnitNo                   := #UnitNo,
           ActRec                   := DB2310.J6FRV1,
           Typ                      := 4,
           FBa                      := #xTmp,
           FBa2                     := #xTmp,
           Out                      := #xTmp);

END_FUNCTION_BLOCK

FUNCTION_BLOCK FB 1311
TITLE =U031: Well Transfer J6
FAMILY : BOTEC_F1
NAME : UniE
VERSION : 1.2


VAR_TEMP
  CIP : BOOL ;	//CIP active
  UNIM : BOOL ;	//Unit Not In Maintenance
  GenRel : BOOL ;	//general OK (emergency and maintenance OK)
  EStopOK : BOOL ;	//emergency OK
  UnitNo : INT ;	//unit number
  xTmp : BOOL ;	//Temporary Bool
  iTmp : INT ;	//Temporary INT
  rTmp : REAL ;	//Temporary REAL
  dTmp : DINT ;	//Temporary DINT (free for general use)
  RetValInt : INT ;	//return value
  DSTUnit : INT ;	//Destination Water Tank
  wRetVal : WORD ;	//return value as word
END_VAR
BEGIN
NETWORK
TITLE =General

      SET   ;
// Simulation ---------------------------------------------------------------
      A     DB1311.DBX 1357.7;
      CC    FB  1319; // "U031Sim"
      A     DB1311.DBX   17.3;
      =     DB1311.DBX 1357.7; //Help bit for simulation

// get unit number ----------------------------------------------------------
      L     DB1310.DBW    0;
      T     #UnitNo;

// communication ------------------------------------------------------------
      UC    FB  1315; // U031Com

NETWORK
TITLE =Sequence organisation

      CLR   ;
      =     M    122.2;

// sequencer ----------------------------------------------------------------
      A     DB1313.DBX   43.1;
      S     DB1313.DBX   97.3;

      CALL FC    40 (
           UnitNo                   := #UnitNo);

END_FUNCTION_BLOCK

FUNCTION_BLOCK FB 1320
TITLE =U032: Well Transfer L6F
FAMILY : BOTEC_F1
NAME : UniA
VERSION : 2.1


VAR_TEMP
  EStopOK : BOOL ;	//auxiliary flag
  CIP : BOOL ;	//CIP Program Selected
  xTmp : BOOL ;	//Temporary Bool(free for general use)
  UnitNo : INT ;	//unit number
  UnitFB : INT ;	//unit expansion FB number
  rTmp : REAL ;	//Temporary REAL (free for general use)
  iTmp : INT ;	//Temporary INT (free for general use)
  dTmp : DINT ;	//Temporary DINT (free for general use)
END_VAR
BEGIN
NETWORK
TITLE =general

      CLR   ;
      =     #xTmp;
      =     #EStopOK;

      L     DB1320.DBW    0;
      T     #UnitNo;
      L     DB1320.DBW    2;
      T     #UnitFB;

NETWORK
TITLE =analog inputs

      NOP   0;
// C_AnI01 AnI 001 spare
      CALL FC    24 (
           UnitNo                   := #UnitNo,
           AnIRec                   := DB2323.C_AnI01,
           ValPer                   := #iTmp);

// QI_CO2_L6F_PH AnI 002
      CALL FC    24 (
           UnitNo                   := #UnitNo,
           AnIRec                   := DB2323.QI_CO2_L6F_PH,
           ValPer                   := IW   210);

// AnI03 AnI 003 spare
      CALL FC    24 (
           UnitNo                   := #UnitNo,
           AnIRec                   := DB2323.AnI03,
           ValPer                   := #iTmp);

NETWORK
TITLE =Universal value

      NOP   0;
// unv001 UnV 001 Process Status
      CALL FC    27 (
           UnitNo                   := #UnitNo,
           UnVRec                   := DB2325.unv001,
           ValExt                   := DB2325.DBD  234);

// unv002 UnV 002 Universal Value 02
      CALL FC    27 (
           UnitNo                   := #UnitNo,
           UnVRec                   := DB2325.unv002,
           ValExt                   := DB2325.DBD  362);

// unv003 UnV 003 Universal Value 03
      CALL FC    27 (
           UnitNo                   := #UnitNo,
           UnVRec                   := DB2325.unv003,
           ValExt                   := DB2325.DBD  490);

// unv004 UnV 004 Universal Value 04
      CALL FC    27 (
           UnitNo                   := #UnitNo,
           UnVRec                   := DB2325.unv004,
           ValExt                   := DB2325.DBD  618);

NETWORK
TITLE =special inputs

      NOP   0;
// SpI01 SpI 001 spare
      CALL FC    14 (
           UnitNo                   := #UnitNo,
           SpIRec                   := DB2321.SpI01,
           SpIBit                   := #xTmp);

// SpI02 SpI 002 spare
      CALL FC    14 (
           UnitNo                   := #UnitNo,
           SpIRec                   := DB2321.SpI02,
           SpIBit                   := #xTmp);

// SpI03 SpI 003 spare
      CALL FC    14 (
           UnitNo                   := #UnitNo,
           SpIRec                   := DB2321.SpI03,
           SpIBit                   := #xTmp);

// SpI04 SpI 004 spare
      CALL FC    14 (
           UnitNo                   := #UnitNo,
           SpIRec                   := DB2321.SpI04,
           SpIBit                   := #xTmp);

NETWORK
TITLE =messages

      NOP   0;
// msg001 Msg 001 Message 01
      CALL FC    16 (
           UnitNo                   := #UnitNo,
           MsgRec                   := DB2327.msg001,
           MsgBit                   := DB2327.DBX   82.7);

// msg002 Msg 002 Message 02
      CALL FC    16 (
           UnitNo                   := #UnitNo,
           MsgRec                   := DB2327.msg002,
           MsgBit                   := DB2327.DBX  142.7);

// msg003 Msg 003 Message 03
      CALL FC    16 (
           UnitNo                   := #UnitNo,
           MsgRec                   := DB2327.msg003,
           MsgBit                   := DB2327.DBX  202.7);

NETWORK
TITLE =controllers

      NOP   0;
// CO2L6FRV1 PID 001 CO2 L6F RV1
      CALL FC    55 (
           UnitNo                   := #UnitNo,
           PIDRec                   := DB2326.CO2L6FRV1,
           SpExt                    := DB2326.DBD  234,
           PVal                     := DB2326.DBD  254,
           OPer                     := PQW  542);

NETWORK
TITLE =unit supply

      UC    FB [#UnitFB];

NETWORK
TITLE =L6F_G1  L6F_G1
// Act 001
// Box           : VS2-BB
// Output address: Q310.0
      CALL FC    70 (
           UnitNo                   := #UnitNo,
           ActRec                   := DB2320.L6F_G1,
           Typ                      := 0,
           FBa                      := #xTmp,
           FBa2                     := I    310.0,
           Out                      := Q    310.0);

NETWORK
TITLE =CO2_L6FV2  Ansteuerung L6FV2
// Act 002
// Box           : CO2 Dosierung
// Output address: Q61.3
      CALL FC    70 (
           UnitNo                   := #UnitNo,
           ActRec                   := DB2320.CO2_L6FV2,
           Typ                      := 0,
           FBa                      := #xTmp,
           FBa2                     := #xTmp,
           Out                      := Q     61.3);

NETWORK
TITLE =CO2_L6FV1  Ansteuerung L6FV1
// Act 003
// Box           : CO2 Dosierung
// Output address: Q60.3
      CALL FC    70 (
           UnitNo                   := #UnitNo,
           ActRec                   := DB2320.CO2_L6FV1,
           Typ                      := 0,
           FBa                      := #xTmp,
           FBa2                     := #xTmp,
           Out                      := Q     60.3);

NETWORK
TITLE =L6FRV1  CO2 L6F RV1
// Act 004
// Box           :
// Input address : #xtmp
// Output address: #xtmp
      CALL FC    70 (
           UnitNo                   := #UnitNo,
           ActRec                   := DB2320.L6FRV1,
           Typ                      := 4,
           FBa                      := #xTmp,
           FBa2                     := #xTmp,
           Out                      := #xTmp);

END_FUNCTION_BLOCK

FUNCTION_BLOCK FB 1321
TITLE =U032: Well Transfer L6F
FAMILY : BOTEC_F1
NAME : UniE
VERSION : 1.2


VAR_TEMP
  CIP : BOOL ;	//CIP active
  UNIM : BOOL ;	//Unit Not In Maintenance
  GenRel : BOOL ;	//general OK (emergency and maintenance OK)
  EStopOK : BOOL ;	//emergency OK
  UnitNo : INT ;	//unit number
  xTmp : BOOL ;	//Temporary Bool
  iTmp : INT ;	//Temporary INT
  rTmp : REAL ;	//Temporary REAL
  dTmp : DINT ;	//Temporary DINT (free for general use)
  RetValInt : INT ;	//return value
END_VAR
BEGIN
NETWORK
TITLE =General

      SET   ;
// Simulation ---------------------------------------------------------------
      A     DB1321.DBX 1357.7;
      CC    FB  1329; // "U032Sim"
      A     DB1321.DBX   17.3;
      =     DB1321.DBX 1357.7; //Help bit for simulation

// get unit number ----------------------------------------------------------
      L     DB1320.DBW    0;
      T     #UnitNo;

// communication ------------------------------------------------------------
      UC    FB  1325; // U032Com

NETWORK
TITLE =Sequence organisation

      CLR   ;
      =     M    122.2;

// sequencer ----------------------------------------------------------------
      A     DB1323.DBX   43.1;
      S     DB1323.DBX   97.3;

      CALL FC    40 (
           UnitNo                   := #UnitNo);

END_FUNCTION_BLOCK

FUNCTION_BLOCK FB 1330
TITLE =U033: Well Transfer B6
FAMILY : BOTEC_F1
NAME : UniA
VERSION : 2.1


VAR_TEMP
  EStopOK : BOOL ;	//auxiliary flag
  CIP : BOOL ;	//CIP Program Selected
  xTmp : BOOL ;	//Temporary Bool(free for general use)
  UnitNo : INT ;	//unit number
  UnitFB : INT ;	//unit expansion FB number
  rTmp : REAL ;	//Temporary REAL (free for general use)
  iTmp : INT ;	//Temporary INT (free for general use)
  dTmp : DINT ;	//Temporary DINT (free for general use)
END_VAR
BEGIN
NETWORK
TITLE =general

      CLR   ;
      =     #xTmp;
      =     #EStopOK;

      L     DB1330.DBW    0;
      T     #UnitNo;
      L     DB1330.DBW    2;
      T     #UnitFB;

NETWORK
TITLE =analog inputs

      NOP   0;
// C_AnI01 AnI 001 spare
      CALL FC    24 (
           UnitNo                   := #UnitNo,
           AnIRec                   := DB2333.C_AnI01,
           ValPer                   := #iTmp);

// QI_CO2_B6_PH AnI 002
      CALL FC    24 (
           UnitNo                   := #UnitNo,
           AnIRec                   := DB2333.QI_CO2_B6_PH,
           ValPer                   := IW   214);

// AnI03 AnI 003 spare
      CALL FC    24 (
           UnitNo                   := #UnitNo,
           AnIRec                   := DB2333.AnI03,
           ValPer                   := #iTmp);

NETWORK
TITLE =Universal value

      NOP   0;
// unv001 UnV 001 Process Status
      CALL FC    27 (
           UnitNo                   := #UnitNo,
           UnVRec                   := DB2335.unv001,
           ValExt                   := DB2335.DBD  234);

// unv002 UnV 002 Universal Value 02
      CALL FC    27 (
           UnitNo                   := #UnitNo,
           UnVRec                   := DB2335.unv002,
           ValExt                   := DB2335.DBD  362);

// unv003 UnV 003 Universal Value 03
      CALL FC    27 (
           UnitNo                   := #UnitNo,
           UnVRec                   := DB2335.unv003,
           ValExt                   := DB2335.DBD  490);

// unv004 UnV 004 Universal Value 04
      CALL FC    27 (
           UnitNo                   := #UnitNo,
           UnVRec                   := DB2335.unv004,
           ValExt                   := DB2335.DBD  618);

NETWORK
TITLE =special inputs

      NOP   0;
// SpI01 SpI 001 spare
      CALL FC    14 (
           UnitNo                   := #UnitNo,
           SpIRec                   := DB2331.SpI01,
           SpIBit                   := #xTmp);

// SpI02 SpI 002 spare
      CALL FC    14 (
           UnitNo                   := #UnitNo,
           SpIRec                   := DB2331.SpI02,
           SpIBit                   := #xTmp);

// SpI03 SpI 003 spare
      CALL FC    14 (
           UnitNo                   := #UnitNo,
           SpIRec                   := DB2331.SpI03,
           SpIBit                   := #xTmp);

// SpI04 SpI 004 spare
      CALL FC    14 (
           UnitNo                   := #UnitNo,
           SpIRec                   := DB2331.SpI04,
           SpIBit                   := #xTmp);

NETWORK
TITLE =messages

      NOP   0;
// msg001 Msg 001 Message 01
      CALL FC    16 (
           UnitNo                   := #UnitNo,
           MsgRec                   := DB2337.msg001,
           MsgBit                   := DB2337.DBX   82.7);

// msg002 Msg 002 Message 02
      CALL FC    16 (
           UnitNo                   := #UnitNo,
           MsgRec                   := DB2337.msg002,
           MsgBit                   := DB2337.DBX  142.7);

// msg003 Msg 003 Message 03
      CALL FC    16 (
           UnitNo                   := #UnitNo,
           MsgRec                   := DB2337.msg003,
           MsgBit                   := DB2337.DBX  202.7);

NETWORK
TITLE =controllers

      NOP   0;
// CO2B6RV1 PID 001 CO2 B6 RV1
      CALL FC    55 (
           UnitNo                   := #UnitNo,
           PIDRec                   := DB2336.CO2B6RV1,
           SpExt                    := DB2336.DBD  234,
           PVal                     := DB2336.DBD  254,
           OPer                     := PQW  546);

NETWORK
TITLE =unit supply

      UC    FB [#UnitFB];

NETWORK
TITLE =B6_G1  B6_G1
// Act 001
// Box           : VS2-BB
// Output address: Q310.1
      CALL FC    70 (
           UnitNo                   := #UnitNo,
           ActRec                   := DB2330.B6_G1,
           Typ                      := 1,
           FBa                      := #xTmp,
           FBa2                     := I    310.1,
           Out                      := Q    310.1);

NETWORK
TITLE =CO2_B6V2  Ansteuerung B6V2
// Act 002
// Box           : CO2 Dosierung
// Output address: Q61.5
      CALL FC    70 (
           UnitNo                   := #UnitNo,
           ActRec                   := DB2330.CO2_B6V2,
           Typ                      := 0,
           FBa                      := #xTmp,
           FBa2                     := #xTmp,
           Out                      := Q     61.5);

NETWORK
TITLE =CO2_B6V1  Ansteuerung B6V1
// Act 003
// Box           : CO2 Dosierung
// Output address: Q60.5
      CALL FC    70 (
           UnitNo                   := #UnitNo,
           ActRec                   := DB2330.CO2_B6V1,
           Typ                      := 0,
           FBa                      := #xTmp,
           FBa2                     := #xTmp,
           Out                      := Q     60.5);

NETWORK
TITLE =B6RV1  CO2 B6 RV1
// Act 004
// Box           :
// Input address : #xtmp
// Output address: #xtmp
      CALL FC    70 (
           UnitNo                   := #UnitNo,
           ActRec                   := DB2330.B6RV1,
           Typ                      := 4,
           FBa                      := #xTmp,
           FBa2                     := #xTmp,
           Out                      := #xTmp);

END_FUNCTION_BLOCK

FUNCTION_BLOCK FB 1331
TITLE =U033: Well Transfer B6
FAMILY : BOTEC_F1
NAME : UniE
VERSION : 1.2


VAR_TEMP
  CIP : BOOL ;	//CIP active
  UNIM : BOOL ;	//Unit Not In Maintenance
  GenRel : BOOL ;	//general OK (emergency and maintenance OK)
  EStopOK : BOOL ;	//emergency OK
  UnitNo : INT ;	//unit number
  xTmp : BOOL ;	//Temporary Bool
  iTmp : INT ;	//Temporary INT
  rTmp : REAL ;	//Temporary REAL
  dTmp : DINT ;	//Temporary DINT (free for general use)
  RetValInt : INT ;	//return value
END_VAR
BEGIN
NETWORK
TITLE =General

      SET   ;
// Simulation ---------------------------------------------------------------
      A     DB1331.DBX 1357.7;
      CC    FB  1339; // "U033Sim"
      A     DB1331.DBX   17.3;
      =     DB1331.DBX 1357.7; //Help bit for simulation

// get unit number ----------------------------------------------------------
      L     DB1330.DBW    0;
      T     #UnitNo;

// communication ------------------------------------------------------------
      UC    FB  1335; // U033Com

NETWORK
TITLE =Sequence organisation

      CLR   ;
      =     M    122.2;

// sequencer ----------------------------------------------------------------
      A     DB1333.DBX   43.1;
      S     DB1333.DBX   97.3;

      CALL FC    40 (
           UnitNo                   := #UnitNo);

END_FUNCTION_BLOCK

FUNCTION_BLOCK FB 1340
TITLE =U034: Well Transfer D6
FAMILY : BOTEC_F1
NAME : UniA
VERSION : 2.1


VAR_TEMP
  EStopOK : BOOL ;	//auxiliary flag
  CIP : BOOL ;	//CIP Program Selected
  xTmp : BOOL ;	//Temporary Bool(free for general use)
  UnitNo : INT ;	//unit number
  UnitFB : INT ;	//unit expansion FB number
  rTmp : REAL ;	//Temporary REAL (free for general use)
  iTmp : INT ;	//Temporary INT (free for general use)
  dTmp : DINT ;	//Temporary DINT (free for general use)
END_VAR
BEGIN
NETWORK
TITLE =general

      CLR   ;
      =     #xTmp;
      =     #EStopOK;

      L     DB1340.DBW    0;
      T     #UnitNo;
      L     DB1340.DBW    2;
      T     #UnitFB;

NETWORK
TITLE =analog inputs

      NOP   0;
// C_AnI01 AnI 001 spare
      CALL FC    24 (
           UnitNo                   := #UnitNo,
           AnIRec                   := DB2343.C_AnI01,
           ValPer                   := #iTmp);

// QI_CO2_D6_PH AnI 002
      CALL FC    24 (
           UnitNo                   := #UnitNo,
           AnIRec                   := DB2343.QI_CO2_D6_PH,
           ValPer                   := IW   212);

// AnI03 AnI 003 spare
      CALL FC    24 (
           UnitNo                   := #UnitNo,
           AnIRec                   := DB2343.AnI03,
           ValPer                   := #iTmp);

NETWORK
TITLE =Universal value

      NOP   0;
// unv001 UnV 001 Process Status
      CALL FC    27 (
           UnitNo                   := #UnitNo,
           UnVRec                   := DB2345.unv001,
           ValExt                   := DB2345.DBD  234);

// unv002 UnV 002 Universal Value 02
      CALL FC    27 (
           UnitNo                   := #UnitNo,
           UnVRec                   := DB2345.unv002,
           ValExt                   := DB2345.DBD  362);

// unv003 UnV 003 Universal Value 03
      CALL FC    27 (
           UnitNo                   := #UnitNo,
           UnVRec                   := DB2345.unv003,
           ValExt                   := DB2345.DBD  490);

// unv004 UnV 004 Universal Value 04
      CALL FC    27 (
           UnitNo                   := #UnitNo,
           UnVRec                   := DB2345.unv004,
           ValExt                   := DB2345.DBD  618);

NETWORK
TITLE =special inputs

      NOP   0;
// SpI01 SpI 001 spare
      CALL FC    14 (
           UnitNo                   := #UnitNo,
           SpIRec                   := DB2341.SpI01,
           SpIBit                   := #xTmp);

// SpI02 SpI 002 spare
      CALL FC    14 (
           UnitNo                   := #UnitNo,
           SpIRec                   := DB2341.SpI02,
           SpIBit                   := #xTmp);

// SpI03 SpI 003 spare
      CALL FC    14 (
           UnitNo                   := #UnitNo,
           SpIRec                   := DB2341.SpI03,
           SpIBit                   := #xTmp);

// SpI04 SpI 004 spare
      CALL FC    14 (
           UnitNo                   := #UnitNo,
           SpIRec                   := DB2341.SpI04,
           SpIBit                   := #xTmp);

NETWORK
TITLE =messages

      NOP   0;
// msg001 Msg 001 Message 01
      CALL FC    16 (
           UnitNo                   := #UnitNo,
           MsgRec                   := DB2347.msg001,
           MsgBit                   := DB2347.DBX   82.7);

// msg002 Msg 002 Message 02
      CALL FC    16 (
           UnitNo                   := #UnitNo,
           MsgRec                   := DB2347.msg002,
           MsgBit                   := DB2347.DBX  142.7);

// msg003 Msg 003 Message 03
      CALL FC    16 (
           UnitNo                   := #UnitNo,
           MsgRec                   := DB2347.msg003,
           MsgBit                   := DB2347.DBX  202.7);

NETWORK
TITLE =controllers

